// ---- VISUs/EtherCAT_Diag2.TcVIS
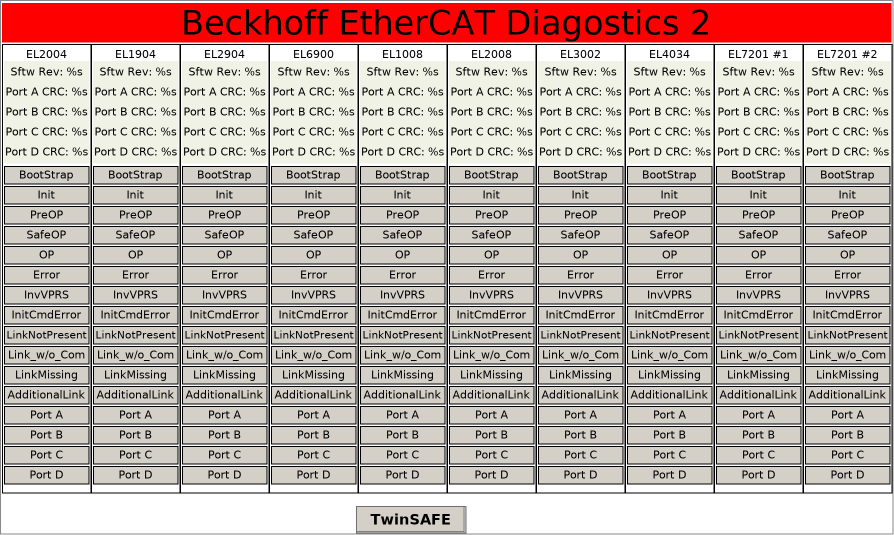
VISUALIZATION EtherCAT_Diag2  // 894x535
    Button (356,506 110x27), "TwinSAFE"
        OnMouseClick: change screen: TwinSAFE
    RoundedRectangle (2,3 889x39), "Beckhoff EtherCAT Diagostics 2"
    Group (2,42 89x451)
        RoundedRectangle (0,2 89x449)
        Label (2,0 85x25), "EL2004"
        Rectangle (2,19 85x22), "Sftw Rev: %s", text variable: g_iHMI_ProdCodeEL2004
        Rectangle (2,39 85x22), "Port A CRC: %s", text variable: g_stHMI_EL2004CrcErrorEx.portA
        Rectangle (2,59 85x22), "Port B CRC: %s", text variable: g_stHMI_EL2004CrcErrorEx.portB
        Rectangle (2,79 85x22), "Port C CRC: %s", text variable: g_stHMI_EL2004CrcErrorEx.portC
        Rectangle (2,99 85x22), "Port D CRC: %s", text variable: g_stHMI_EL2004CrcErrorEx.portD
        Rectangle (2,124 85x18), "BootStrap", colour toggle: g_stHMI_EL2004EcSlaveStateBits.bBootStrap
        Rectangle (2,144 85x18), "Init", colour toggle: g_stHMI_EL2004EcSlaveStateBits.bInit
        Rectangle (2,164 85x18), "PreOP", colour toggle: g_stHMI_EL2004EcSlaveStateBits.bPreop
        Rectangle (2,184 85x18), "SafeOP", colour toggle: g_stHMI_EL2004EcSlaveStateBits.bSafeOp
        Rectangle (2,204 85x18), "OP", colour toggle: g_stHMI_EL2004EcSlaveStateBits.bOp
        Rectangle (2,224 85x18), "Error", colour toggle: g_stHMI_EL2004EcSlaveStateBits.bError
        Rectangle (2,244 85x18), "InvVPRS", colour toggle: g_stHMI_EL2004EcSlaveStateBits.bInvVPRS
        Rectangle (2,264 85x18), "InitCmdError", colour toggle: g_stHMI_EL2004EcSlaveStateBits.bInitCmdError
        Rectangle (2,284 85x18), "LinkNotPresent", colour toggle: g_stHMI_EL2004EcSlaveStateBits.bLinkNotPresent
        Rectangle (2,304 85x18), "Link_w/o_Com", colour toggle: g_stHMI_EL2004EcSlaveStateBits.bLinkWithoutComm
        Rectangle (2,324 85x18), "LinkMissing", colour toggle: g_stHMI_EL2004EcSlaveStateBits.bLinkMissing
        Rectangle (2,344 85x18), "AdditionalLink", colour toggle: g_stHMI_EL2004EcSlaveStateBits.bAdditionalLink
        Rectangle (2,364 85x18), "Port A", colour toggle: g_stHMI_EL2004EcSlaveStateBits.bPortA
        Rectangle (2,384 85x18), "Port B", colour toggle: g_stHMI_EL2004EcSlaveStateBits.bPortB
        Rectangle (2,404 85x18), "Port C", colour toggle: g_stHMI_EL2004EcSlaveStateBits.bPortC
        Rectangle (2,424 85x18), "Port D", colour toggle: g_stHMI_EL2004EcSlaveStateBits.bPortD
    Group (91,42 89x451)
        RoundedRectangle (0,2 89x449)
        Label (2,0 85x25), "EL1904"
        Rectangle (2,19 85x22), "Sftw Rev: %s", text variable: g_iHMI_ProdCodeEL1904
        Rectangle (2,39 85x22), "Port A CRC: %s", text variable: g_stHMI_EL1904CrcErrorEx.portA
        Rectangle (2,59 85x22), "Port B CRC: %s", text variable: g_stHMI_EL1904CrcErrorEx.portB
        Rectangle (2,79 85x22), "Port C CRC: %s", text variable: g_stHMI_EL1904CrcErrorEx.portC
        Rectangle (2,99 85x22), "Port D CRC: %s", text variable: g_stHMI_EL1904CrcErrorEx.portD
        Rectangle (2,124 85x18), "BootStrap", colour toggle: g_stHMI_EL1904EcSlaveStateBits.bBootStrap
        Rectangle (2,144 85x18), "Init", colour toggle: g_stHMI_EL1904EcSlaveStateBits.bInit
        Rectangle (2,164 85x18), "PreOP", colour toggle: g_stHMI_EL1904EcSlaveStateBits.bPreop
        Rectangle (2,184 85x18), "SafeOP", colour toggle: g_stHMI_EL1904EcSlaveStateBits.bSafeOp
        Rectangle (2,204 85x18), "OP", colour toggle: g_stHMI_EL1904EcSlaveStateBits.bOp
        Rectangle (2,224 85x18), "Error", colour toggle: g_stHMI_EL1904EcSlaveStateBits.bError
        Rectangle (2,244 85x18), "InvVPRS", colour toggle: g_stHMI_EL1904EcSlaveStateBits.bInvVPRS
        Rectangle (2,264 85x18), "InitCmdError", colour toggle: g_stHMI_EL1904EcSlaveStateBits.bInitCmdError
        Rectangle (2,284 85x18), "LinkNotPresent", colour toggle: g_stHMI_EL1904EcSlaveStateBits.bLinkNotPresent
        Rectangle (2,304 85x18), "Link_w/o_Com", colour toggle: g_stHMI_EL1904EcSlaveStateBits.bLinkWithoutComm
        Rectangle (2,324 85x18), "LinkMissing", colour toggle: g_stHMI_EL1904EcSlaveStateBits.bLinkMissing
        Rectangle (2,344 85x18), "AdditionalLink", colour toggle: g_stHMI_EL1904EcSlaveStateBits.bAdditionalLink
        Rectangle (2,364 85x18), "Port A", colour toggle: g_stHMI_EL1904EcSlaveStateBits.bPortA
        Rectangle (2,384 85x18), "Port B", colour toggle: g_stHMI_EL1904EcSlaveStateBits.bPortB
        Rectangle (2,404 85x18), "Port C", colour toggle: g_stHMI_EL1904EcSlaveStateBits.bPortC
        Rectangle (2,424 85x18), "Port D", colour toggle: g_stHMI_EL1904EcSlaveStateBits.bPortD
    Group (180,42 89x451)
        RoundedRectangle (0,2 89x449)
        Label (2,0 85x25), "EL2904"
        Rectangle (2,19 85x22), "Sftw Rev: %s", text variable: g_iHMI_ProdCodeEL2904
        Rectangle (2,39 85x22), "Port A CRC: %s", text variable: g_stHMI_EL2904CrcErrorEx.portA
        Rectangle (2,59 85x22), "Port B CRC: %s", text variable: g_stHMI_EL2904CrcErrorEx.portB
        Rectangle (2,79 85x22), "Port C CRC: %s", text variable: g_stHMI_EL2904CrcErrorEx.portC
        Rectangle (2,99 85x22), "Port D CRC: %s", text variable: g_stHMI_EL2904CrcErrorEx.portD
        Rectangle (2,124 85x18), "BootStrap", colour toggle: g_stHMI_EL2904EcSlaveStateBits.bBootStrap
        Rectangle (2,144 85x18), "Init", colour toggle: g_stHMI_EL2904EcSlaveStateBits.bInit
        Rectangle (2,164 85x18), "PreOP", colour toggle: g_stHMI_EL2904EcSlaveStateBits.bPreop
        Rectangle (2,184 85x18), "SafeOP", colour toggle: g_stHMI_EL2904EcSlaveStateBits.bSafeOp
        Rectangle (2,204 85x18), "OP", colour toggle: g_stHMI_EL2904EcSlaveStateBits.bOp
        Rectangle (2,224 85x18), "Error", colour toggle: g_stHMI_EL2904EcSlaveStateBits.bError
        Rectangle (2,244 85x18), "InvVPRS", colour toggle: g_stHMI_EL2904EcSlaveStateBits.bInvVPRS
        Rectangle (2,264 85x18), "InitCmdError", colour toggle: g_stHMI_EL2904EcSlaveStateBits.bInitCmdError
        Rectangle (2,284 85x18), "LinkNotPresent", colour toggle: g_stHMI_EL2904EcSlaveStateBits.bLinkNotPresent
        Rectangle (2,304 85x18), "Link_w/o_Com", colour toggle: g_stHMI_EL2904EcSlaveStateBits.bLinkWithoutComm
        Rectangle (2,324 85x18), "LinkMissing", colour toggle: g_stHMI_EL2904EcSlaveStateBits.bLinkMissing
        Rectangle (2,344 85x18), "AdditionalLink", colour toggle: g_stHMI_EL2904EcSlaveStateBits.bAdditionalLink
        Rectangle (2,364 85x18), "Port A", colour toggle: g_stHMI_EL2904EcSlaveStateBits.bPortA
        Rectangle (2,384 85x18), "Port B", colour toggle: g_stHMI_EL2904EcSlaveStateBits.bPortB
        Rectangle (2,404 85x18), "Port C", colour toggle: g_stHMI_EL2904EcSlaveStateBits.bPortC
        Rectangle (2,424 85x18), "Port D", colour toggle: g_stHMI_EL2904EcSlaveStateBits.bPortD
    Group (269,42 89x451)
        RoundedRectangle (0,2 89x449)
        Label (2,0 85x25), "EL6900"
        Rectangle (2,19 85x22), "Sftw Rev: %s", text variable: g_iHMI_ProdCodeEL6900
        Rectangle (2,39 85x22), "Port A CRC: %s", text variable: g_stHMI_EL6900CrcErrorEx.portA
        Rectangle (2,59 85x22), "Port B CRC: %s", text variable: g_stHMI_EL6900CrcErrorEx.portB
        Rectangle (2,79 85x22), "Port C CRC: %s", text variable: g_stHMI_EL6900CrcErrorEx.portC
        Rectangle (2,99 85x22), "Port D CRC: %s", text variable: g_stHMI_EL6900CrcErrorEx.portD
        Rectangle (2,124 85x18), "BootStrap", colour toggle: g_stHMI_EL6900EcSlaveStateBits.bBootStrap
        Rectangle (2,144 85x18), "Init", colour toggle: g_stHMI_EL6900EcSlaveStateBits.bInit
        Rectangle (2,164 85x18), "PreOP", colour toggle: g_stHMI_EL6900EcSlaveStateBits.bPreop
        Rectangle (2,184 85x18), "SafeOP", colour toggle: g_stHMI_EL6900EcSlaveStateBits.bSafeOp
        Rectangle (2,204 85x18), "OP", colour toggle: g_stHMI_EL6900EcSlaveStateBits.bOp
        Rectangle (2,224 85x18), "Error", colour toggle: g_stHMI_EL6900EcSlaveStateBits.bError
        Rectangle (2,244 85x18), "InvVPRS", colour toggle: g_stHMI_EL6900EcSlaveStateBits.bInvVPRS
        Rectangle (2,264 85x18), "InitCmdError", colour toggle: g_stHMI_EL6900EcSlaveStateBits.bInitCmdError
        Rectangle (2,284 85x18), "LinkNotPresent", colour toggle: g_stHMI_EL6900EcSlaveStateBits.bLinkNotPresent
        Rectangle (2,304 85x18), "Link_w/o_Com", colour toggle: g_stHMI_EL6900EcSlaveStateBits.bLinkWithoutComm
        Rectangle (2,324 85x18), "LinkMissing", colour toggle: g_stHMI_EL6900EcSlaveStateBits.bLinkMissing
        Rectangle (2,344 85x18), "AdditionalLink", colour toggle: g_stHMI_EL6900EcSlaveStateBits.bAdditionalLink
        Rectangle (2,364 85x18), "Port A", colour toggle: g_stHMI_EL6900EcSlaveStateBits.bPortA
        Rectangle (2,384 85x18), "Port B", colour toggle: g_stHMI_EL6900EcSlaveStateBits.bPortB
        Rectangle (2,404 85x18), "Port C", colour toggle: g_stHMI_EL6900EcSlaveStateBits.bPortC
        Rectangle (2,424 85x18), "Port D", colour toggle: g_stHMI_EL6900EcSlaveStateBits.bPortD
    Group (358,42 89x451)
        RoundedRectangle (0,2 89x449)
        Label (2,0 85x25), "EL1008"
        Rectangle (2,19 85x22), "Sftw Rev: %s", text variable: g_iHMI_ProdCodeEL1008
        Rectangle (2,39 85x22), "Port A CRC: %s", text variable: g_stHMI_EL1008CrcErrorEx.portA
        Rectangle (2,59 85x22), "Port B CRC: %s", text variable: g_stHMI_EL1008CrcErrorEx.portB
        Rectangle (2,79 85x22), "Port C CRC: %s", text variable: g_stHMI_EL1008CrcErrorEx.portC
        Rectangle (2,99 85x22), "Port D CRC: %s", text variable: g_stHMI_EL1008CrcErrorEx.portD
        Rectangle (2,124 85x18), "BootStrap", colour toggle: g_stHMI_EL1008EcSlaveStateBits.bBootStrap
        Rectangle (2,144 85x18), "Init", colour toggle: g_stHMI_EL1008EcSlaveStateBits.bInit
        Rectangle (2,164 85x18), "PreOP", colour toggle: g_stHMI_EL1008EcSlaveStateBits.bPreop
        Rectangle (2,184 85x18), "SafeOP", colour toggle: g_stHMI_EL1008EcSlaveStateBits.bSafeOp
        Rectangle (2,204 85x18), "OP", colour toggle: g_stHMI_EL1008EcSlaveStateBits.bOp
        Rectangle (2,224 85x18), "Error", colour toggle: g_stHMI_EL1008EcSlaveStateBits.bError
        Rectangle (2,244 85x18), "InvVPRS", colour toggle: g_stHMI_EL1008EcSlaveStateBits.bInvVPRS
        Rectangle (2,264 85x18), "InitCmdError", colour toggle: g_stHMI_EL1008EcSlaveStateBits.bInitCmdError
        Rectangle (2,284 85x18), "LinkNotPresent", colour toggle: g_stHMI_EL1008EcSlaveStateBits.bLinkNotPresent
        Rectangle (2,304 85x18), "Link_w/o_Com", colour toggle: g_stHMI_EL1008EcSlaveStateBits.bLinkWithoutComm
        Rectangle (2,324 85x18), "LinkMissing", colour toggle: g_stHMI_EL1008EcSlaveStateBits.bLinkMissing
        Rectangle (2,344 85x18), "AdditionalLink", colour toggle: g_stHMI_EL1008EcSlaveStateBits.bAdditionalLink
        Rectangle (2,364 85x18), "Port A", colour toggle: g_stHMI_EL1008EcSlaveStateBits.bPortA
        Rectangle (2,384 85x18), "Port B", colour toggle: g_stHMI_EL1008EcSlaveStateBits.bPortB
        Rectangle (2,404 85x18), "Port C", colour toggle: g_stHMI_EL1008EcSlaveStateBits.bPortC
        Rectangle (2,424 85x18), "Port D", colour toggle: g_stHMI_EL1008EcSlaveStateBits.bPortD
    Group (447,42 89x451)
        RoundedRectangle (0,2 89x449)
        Label (2,0 85x25), "EL2008"
        Rectangle (2,19 85x22), "Sftw Rev: %s", text variable: g_iHMI_ProdCodeEL2008
        Rectangle (2,39 85x22), "Port A CRC: %s", text variable: g_stHMI_EL2008CrcErrorEx.portA
        Rectangle (2,59 85x22), "Port B CRC: %s", text variable: g_stHMI_EL2008CrcErrorEx.portB
        Rectangle (2,79 85x22), "Port C CRC: %s", text variable: g_stHMI_EL2008CrcErrorEx.portC
        Rectangle (2,99 85x22), "Port D CRC: %s", text variable: g_stHMI_EL2008CrcErrorEx.portD
        Rectangle (2,124 85x18), "BootStrap", colour toggle: g_stHMI_EL2008EcSlaveStateBits.bBootStrap
        Rectangle (2,144 85x18), "Init", colour toggle: g_stHMI_EL2008EcSlaveStateBits.bInit
        Rectangle (2,164 85x18), "PreOP", colour toggle: g_stHMI_EL2008EcSlaveStateBits.bPreop
        Rectangle (2,184 85x18), "SafeOP", colour toggle: g_stHMI_EL2008EcSlaveStateBits.bSafeOp
        Rectangle (2,204 85x18), "OP", colour toggle: g_stHMI_EL2008EcSlaveStateBits.bOp
        Rectangle (2,224 85x18), "Error", colour toggle: g_stHMI_EL2008EcSlaveStateBits.bError
        Rectangle (2,244 85x18), "InvVPRS", colour toggle: g_stHMI_EL2008EcSlaveStateBits.bInvVPRS
        Rectangle (2,264 85x18), "InitCmdError", colour toggle: g_stHMI_EL2008EcSlaveStateBits.bInitCmdError
        Rectangle (2,284 85x18), "LinkNotPresent", colour toggle: g_stHMI_EL2008EcSlaveStateBits.bLinkNotPresent
        Rectangle (2,304 85x18), "Link_w/o_Com", colour toggle: g_stHMI_EL2008EcSlaveStateBits.bLinkWithoutComm
        Rectangle (2,324 85x18), "LinkMissing", colour toggle: g_stHMI_EL2008EcSlaveStateBits.bLinkMissing
        Rectangle (2,344 85x18), "AdditionalLink", colour toggle: g_stHMI_EL2008EcSlaveStateBits.bAdditionalLink
        Rectangle (2,364 85x18), "Port A", colour toggle: g_stHMI_EL2008EcSlaveStateBits.bPortA
        Rectangle (2,384 85x18), "Port B", colour toggle: g_stHMI_EL2008EcSlaveStateBits.bPortB
        Rectangle (2,404 85x18), "Port C", colour toggle: g_stHMI_EL2008EcSlaveStateBits.bPortC
        Rectangle (2,424 85x18), "Port D", colour toggle: g_stHMI_EL2008EcSlaveStateBits.bPortD
    Group (536,42 89x451)
        RoundedRectangle (0,2 89x449)
        Label (2,0 85x25), "EL3002"
        Rectangle (2,19 85x22), "Sftw Rev: %s", text variable: g_iHMI_ProdCodeEL3002
        Rectangle (2,39 85x22), "Port A CRC: %s", text variable: g_stHMI_EL3002CrcErrorEx.portA
        Rectangle (2,59 85x22), "Port B CRC: %s", text variable: g_stHMI_EL3002CrcErrorEx.portB
        Rectangle (2,79 85x22), "Port C CRC: %s", text variable: g_stHMI_EL3002CrcErrorEx.portC
        Rectangle (2,99 85x22), "Port D CRC: %s", text variable: g_stHMI_EL3002CrcErrorEx.portD
        Rectangle (2,124 85x18), "BootStrap", colour toggle: g_stHMI_EL3002EcSlaveStateBits.bBootStrap
        Rectangle (2,144 85x18), "Init", colour toggle: g_stHMI_EL3002EcSlaveStateBits.bInit
        Rectangle (2,164 85x18), "PreOP", colour toggle: g_stHMI_EL3002EcSlaveStateBits.bPreop
        Rectangle (2,184 85x18), "SafeOP", colour toggle: g_stHMI_EL3002EcSlaveStateBits.bSafeOp
        Rectangle (2,204 85x18), "OP", colour toggle: g_stHMI_EL3002EcSlaveStateBits.bOp
        Rectangle (2,224 85x18), "Error", colour toggle: g_stHMI_EL3002EcSlaveStateBits.bError
        Rectangle (2,244 85x18), "InvVPRS", colour toggle: g_stHMI_EL3002EcSlaveStateBits.bInvVPRS
        Rectangle (2,264 85x18), "InitCmdError", colour toggle: g_stHMI_EL3002EcSlaveStateBits.bInitCmdError
        Rectangle (2,284 85x18), "LinkNotPresent", colour toggle: g_stHMI_EL3002EcSlaveStateBits.bLinkNotPresent
        Rectangle (2,304 85x18), "Link_w/o_Com", colour toggle: g_stHMI_EL3002EcSlaveStateBits.bLinkWithoutComm
        Rectangle (2,324 85x18), "LinkMissing", colour toggle: g_stHMI_EL3002EcSlaveStateBits.bLinkMissing
        Rectangle (2,344 85x18), "AdditionalLink", colour toggle: g_stHMI_EL3002EcSlaveStateBits.bAdditionalLink
        Rectangle (2,364 85x18), "Port A", colour toggle: g_stHMI_EL3002EcSlaveStateBits.bPortA
        Rectangle (2,384 85x18), "Port B", colour toggle: g_stHMI_EL3002EcSlaveStateBits.bPortB
        Rectangle (2,404 85x18), "Port C", colour toggle: g_stHMI_EL3002EcSlaveStateBits.bPortC
        Rectangle (2,424 85x18), "Port D", colour toggle: g_stHMI_EL3002EcSlaveStateBits.bPortD
    Group (625,42 89x451)
        RoundedRectangle (0,2 89x449)
        Label (2,0 85x25), "EL4034"
        Rectangle (2,19 85x22), "Sftw Rev: %s", text variable: g_iHMI_ProdCodeEL4034
        Rectangle (2,39 85x22), "Port A CRC: %s", text variable: g_stHMI_EL4034CrcErrorEx.portA
        Rectangle (2,59 85x22), "Port B CRC: %s", text variable: g_stHMI_EL4034CrcErrorEx.portB
        Rectangle (2,79 85x22), "Port C CRC: %s", text variable: g_stHMI_EL4034CrcErrorEx.portC
        Rectangle (2,99 85x22), "Port D CRC: %s", text variable: g_stHMI_EL4034CrcErrorEx.portD
        Rectangle (2,124 85x18), "BootStrap", colour toggle: g_stHMI_EL4034EcSlaveStateBits.bBootStrap
        Rectangle (2,144 85x18), "Init", colour toggle: g_stHMI_EL4034EcSlaveStateBits.bInit
        Rectangle (2,164 85x18), "PreOP", colour toggle: g_stHMI_EL4034EcSlaveStateBits.bPreop
        Rectangle (2,184 85x18), "SafeOP", colour toggle: g_stHMI_EL4034EcSlaveStateBits.bSafeOp
        Rectangle (2,204 85x18), "OP", colour toggle: g_stHMI_EL4034EcSlaveStateBits.bOp
        Rectangle (2,224 85x18), "Error", colour toggle: g_stHMI_EL4034EcSlaveStateBits.bError
        Rectangle (2,244 85x18), "InvVPRS", colour toggle: g_stHMI_EL4034EcSlaveStateBits.bInvVPRS
        Rectangle (2,264 85x18), "InitCmdError", colour toggle: g_stHMI_EL4034EcSlaveStateBits.bInitCmdError
        Rectangle (2,284 85x18), "LinkNotPresent", colour toggle: g_stHMI_EL4034EcSlaveStateBits.bLinkNotPresent
        Rectangle (2,304 85x18), "Link_w/o_Com", colour toggle: g_stHMI_EL4034EcSlaveStateBits.bLinkWithoutComm
        Rectangle (2,324 85x18), "LinkMissing", colour toggle: g_stHMI_EL4034EcSlaveStateBits.bLinkMissing
        Rectangle (2,344 85x18), "AdditionalLink", colour toggle: g_stHMI_EL4034EcSlaveStateBits.bAdditionalLink
        Rectangle (2,364 85x18), "Port A", colour toggle: g_stHMI_EL4034EcSlaveStateBits.bPortA
        Rectangle (2,384 85x18), "Port B", colour toggle: g_stHMI_EL4034EcSlaveStateBits.bPortB
        Rectangle (2,404 85x18), "Port C", colour toggle: g_stHMI_EL4034EcSlaveStateBits.bPortC
        Rectangle (2,424 85x18), "Port D", colour toggle: g_stHMI_EL4034EcSlaveStateBits.bPortD
    Group (714,42 89x451)
        RoundedRectangle (0,2 89x449)
        Label (2,0 85x25), "EL7201 #1"
        Rectangle (2,19 85x22), "Sftw Rev: %s", text variable: g_iHMI_ProdCodeEL7201_1
        Rectangle (2,39 85x22), "Port A CRC: %s", text variable: g_stHMI_EL7201_1CrcErrorEx.portA
        Rectangle (2,59 85x22), "Port B CRC: %s", text variable: g_stHMI_EL7201_1CrcErrorEx.portB
        Rectangle (2,79 85x22), "Port C CRC: %s", text variable: g_stHMI_EL7201_1CrcErrorEx.portC
        Rectangle (2,99 85x22), "Port D CRC: %s", text variable: g_stHMI_EL7201_1CrcErrorEx.portD
        Rectangle (2,124 85x18), "BootStrap", colour toggle: g_stHMI_EL7201_1EcSlaveStateBits.bBootStrap
        Rectangle (2,144 85x18), "Init", colour toggle: g_stHMI_EL7201_1EcSlaveStateBits.bInit
        Rectangle (2,164 85x18), "PreOP", colour toggle: g_stHMI_EL7201_1EcSlaveStateBits.bPreop
        Rectangle (2,184 85x18), "SafeOP", colour toggle: g_stHMI_EL7201_1EcSlaveStateBits.bSafeOp
        Rectangle (2,204 85x18), "OP", colour toggle: g_stHMI_EL7201_1EcSlaveStateBits.bOp
        Rectangle (2,224 85x18), "Error", colour toggle: g_stHMI_EL7201_1EcSlaveStateBits.bError
        Rectangle (2,244 85x18), "InvVPRS", colour toggle: g_stHMI_EL7201_1EcSlaveStateBits.bInvVPRS
        Rectangle (2,264 85x18), "InitCmdError", colour toggle: g_stHMI_EL7201_1EcSlaveStateBits.bInitCmdError
        Rectangle (2,284 85x18), "LinkNotPresent", colour toggle: g_stHMI_EL7201_1EcSlaveStateBits.bLinkNotPresent
        Rectangle (2,304 85x18), "Link_w/o_Com", colour toggle: g_stHMI_EL7201_1EcSlaveStateBits.bLinkWithoutComm
        Rectangle (2,324 85x18), "LinkMissing", colour toggle: g_stHMI_EL7201_1EcSlaveStateBits.bLinkMissing
        Rectangle (2,344 85x18), "AdditionalLink", colour toggle: g_stHMI_EL7201_1EcSlaveStateBits.bAdditionalLink
        Rectangle (2,364 85x18), "Port A", colour toggle: g_stHMI_EL7201_1EcSlaveStateBits.bPortA
        Rectangle (2,384 85x18), "Port B", colour toggle: g_stHMI_EL7201_1EcSlaveStateBits.bPortB
        Rectangle (2,404 85x18), "Port C", colour toggle: g_stHMI_EL7201_1EcSlaveStateBits.bPortC
        Rectangle (2,424 85x18), "Port D", colour toggle: g_stHMI_EL7201_1EcSlaveStateBits.bPortD
    Group (803,42 89x451)
        RoundedRectangle (0,2 89x449)
        Label (2,0 85x25), "EL7201 #2"
        Rectangle (2,19 85x22), "Sftw Rev: %s", text variable: g_iHMI_ProdCodeEL7201_2
        Rectangle (2,39 85x22), "Port A CRC: %s", text variable: g_stHMI_EL7201_2CrcErrorEx.portA
        Rectangle (2,59 85x22), "Port B CRC: %s", text variable: g_stHMI_EL7201_2CrcErrorEx.portB
        Rectangle (2,79 85x22), "Port C CRC: %s", text variable: g_stHMI_EL7201_2CrcErrorEx.portC
        Rectangle (2,99 85x22), "Port D CRC: %s", text variable: g_stHMI_EL7201_2CrcErrorEx.portD
        Rectangle (2,124 85x18), "BootStrap", colour toggle: g_stHMI_EL7201_2EcSlaveStateBits.bBootStrap
        Rectangle (2,144 85x18), "Init", colour toggle: g_stHMI_EL7201_2EcSlaveStateBits.bInit
        Rectangle (2,164 85x18), "PreOP", colour toggle: g_stHMI_EL7201_2EcSlaveStateBits.bPreop
        Rectangle (2,184 85x18), "SafeOP", colour toggle: g_stHMI_EL7201_2EcSlaveStateBits.bSafeOp
        Rectangle (2,204 85x18), "OP", colour toggle: g_stHMI_EL7201_2EcSlaveStateBits.bOp
        Rectangle (2,224 85x18), "Error", colour toggle: g_stHMI_EL7201_2EcSlaveStateBits.bError
        Rectangle (2,244 85x18), "InvVPRS", colour toggle: g_stHMI_EL7201_2EcSlaveStateBits.bInvVPRS
        Rectangle (2,264 85x18), "InitCmdError", colour toggle: g_stHMI_EL7201_2EcSlaveStateBits.bInitCmdError
        Rectangle (2,284 85x18), "LinkNotPresent", colour toggle: g_stHMI_EL7201_2EcSlaveStateBits.bLinkNotPresent
        Rectangle (2,304 85x18), "Link_w/o_Com", colour toggle: g_stHMI_EL7201_2EcSlaveStateBits.bLinkWithoutComm
        Rectangle (2,324 85x18), "LinkMissing", colour toggle: g_stHMI_EL7201_2EcSlaveStateBits.bLinkMissing
        Rectangle (2,344 85x18), "AdditionalLink", colour toggle: g_stHMI_EL7201_2EcSlaveStateBits.bAdditionalLink
        Rectangle (2,364 85x18), "Port A", colour toggle: g_stHMI_EL7201_2EcSlaveStateBits.bPortA
        Rectangle (2,384 85x18), "Port B", colour toggle: g_stHMI_EL7201_2EcSlaveStateBits.bPortB
        Rectangle (2,404 85x18), "Port C", colour toggle: g_stHMI_EL7201_2EcSlaveStateBits.bPortC
        Rectangle (2,424 85x18), "Port D", colour toggle: g_stHMI_EL7201_2EcSlaveStateBits.bPortD
END_VISUALIZATION

// ---- VISUs/EtherCAT_Diag2.TcVIS
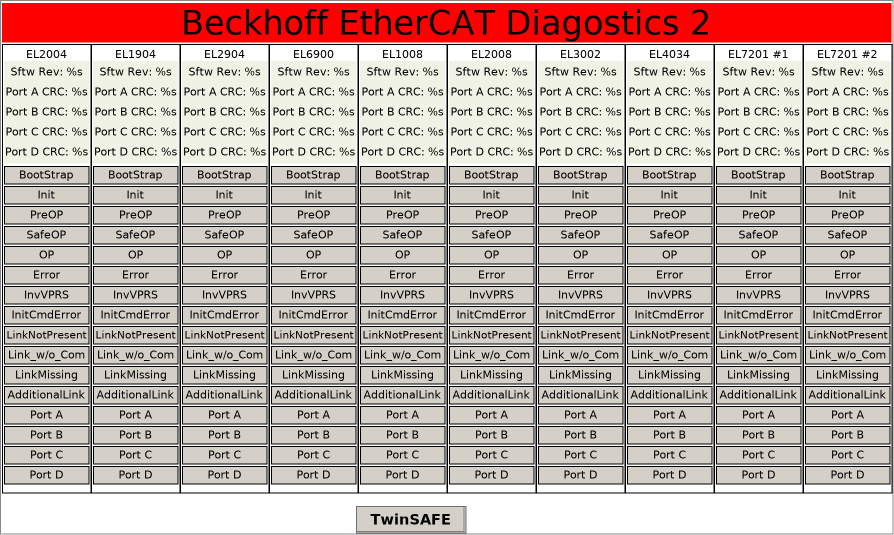
VISUALIZATION EtherCAT_Diag2  // 894x535
    Button (356,506 110x27), "TwinSAFE"
        OnMouseClick: change screen: TwinSAFE
    RoundedRectangle (2,3 889x39), "Beckhoff EtherCAT Diagostics 2"
    Group (2,42 89x451)
        RoundedRectangle (0,2 89x449)
        Label (2,0 85x25), "EL2004"
        Rectangle (2,19 85x22), "Sftw Rev: %s", text variable: g_iHMI_ProdCodeEL2004
        Rectangle (2,39 85x22), "Port A CRC: %s", text variable: g_stHMI_EL2004CrcErrorEx.portA
        Rectangle (2,59 85x22), "Port B CRC: %s", text variable: g_stHMI_EL2004CrcErrorEx.portB
        Rectangle (2,79 85x22), "Port C CRC: %s", text variable: g_stHMI_EL2004CrcErrorEx.portC
        Rectangle (2,99 85x22), "Port D CRC: %s", text variable: g_stHMI_EL2004CrcErrorEx.portD
        Rectangle (2,124 85x18), "BootStrap", colour toggle: g_stHMI_EL2004EcSlaveStateBits.bBootStrap
        Rectangle (2,144 85x18), "Init", colour toggle: g_stHMI_EL2004EcSlaveStateBits.bInit
        Rectangle (2,164 85x18), "PreOP", colour toggle: g_stHMI_EL2004EcSlaveStateBits.bPreop
        Rectangle (2,184 85x18), "SafeOP", colour toggle: g_stHMI_EL2004EcSlaveStateBits.bSafeOp
        Rectangle (2,204 85x18), "OP", colour toggle: g_stHMI_EL2004EcSlaveStateBits.bOp
        Rectangle (2,224 85x18), "Error", colour toggle: g_stHMI_EL2004EcSlaveStateBits.bError
        Rectangle (2,244 85x18), "InvVPRS", colour toggle: g_stHMI_EL2004EcSlaveStateBits.bInvVPRS
        Rectangle (2,264 85x18), "InitCmdError", colour toggle: g_stHMI_EL2004EcSlaveStateBits.bInitCmdError
        Rectangle (2,284 85x18), "LinkNotPresent", colour toggle: g_stHMI_EL2004EcSlaveStateBits.bLinkNotPresent
        Rectangle (2,304 85x18), "Link_w/o_Com", colour toggle: g_stHMI_EL2004EcSlaveStateBits.bLinkWithoutComm
        Rectangle (2,324 85x18), "LinkMissing", colour toggle: g_stHMI_EL2004EcSlaveStateBits.bLinkMissing
        Rectangle (2,344 85x18), "AdditionalLink", colour toggle: g_stHMI_EL2004EcSlaveStateBits.bAdditionalLink
        Rectangle (2,364 85x18), "Port A", colour toggle: g_stHMI_EL2004EcSlaveStateBits.bPortA
        Rectangle (2,384 85x18), "Port B", colour toggle: g_stHMI_EL2004EcSlaveStateBits.bPortB
        Rectangle (2,404 85x18), "Port C", colour toggle: g_stHMI_EL2004EcSlaveStateBits.bPortC
        Rectangle (2,424 85x18), "Port D", colour toggle: g_stHMI_EL2004EcSlaveStateBits.bPortD
    Group (91,42 89x451)
        RoundedRectangle (0,2 89x449)
        Label (2,0 85x25), "EL1904"
        Rectangle (2,19 85x22), "Sftw Rev: %s", text variable: g_iHMI_ProdCodeEL1904
        Rectangle (2,39 85x22), "Port A CRC: %s", text variable: g_stHMI_EL1904CrcErrorEx.portA
        Rectangle (2,59 85x22), "Port B CRC: %s", text variable: g_stHMI_EL1904CrcErrorEx.portB
        Rectangle (2,79 85x22), "Port C CRC: %s", text variable: g_stHMI_EL1904CrcErrorEx.portC
        Rectangle (2,99 85x22), "Port D CRC: %s", text variable: g_stHMI_EL1904CrcErrorEx.portD
        Rectangle (2,124 85x18), "BootStrap", colour toggle: g_stHMI_EL1904EcSlaveStateBits.bBootStrap
        Rectangle (2,144 85x18), "Init", colour toggle: g_stHMI_EL1904EcSlaveStateBits.bInit
        Rectangle (2,164 85x18), "PreOP", colour toggle: g_stHMI_EL1904EcSlaveStateBits.bPreop
        Rectangle (2,184 85x18), "SafeOP", colour toggle: g_stHMI_EL1904EcSlaveStateBits.bSafeOp
        Rectangle (2,204 85x18), "OP", colour toggle: g_stHMI_EL1904EcSlaveStateBits.bOp
        Rectangle (2,224 85x18), "Error", colour toggle: g_stHMI_EL1904EcSlaveStateBits.bError
        Rectangle (2,244 85x18), "InvVPRS", colour toggle: g_stHMI_EL1904EcSlaveStateBits.bInvVPRS
        Rectangle (2,264 85x18), "InitCmdError", colour toggle: g_stHMI_EL1904EcSlaveStateBits.bInitCmdError
        Rectangle (2,284 85x18), "LinkNotPresent", colour toggle: g_stHMI_EL1904EcSlaveStateBits.bLinkNotPresent
        Rectangle (2,304 85x18), "Link_w/o_Com", colour toggle: g_stHMI_EL1904EcSlaveStateBits.bLinkWithoutComm
        Rectangle (2,324 85x18), "LinkMissing", colour toggle: g_stHMI_EL1904EcSlaveStateBits.bLinkMissing
        Rectangle (2,344 85x18), "AdditionalLink", colour toggle: g_stHMI_EL1904EcSlaveStateBits.bAdditionalLink
        Rectangle (2,364 85x18), "Port A", colour toggle: g_stHMI_EL1904EcSlaveStateBits.bPortA
        Rectangle (2,384 85x18), "Port B", colour toggle: g_stHMI_EL1904EcSlaveStateBits.bPortB
        Rectangle (2,404 85x18), "Port C", colour toggle: g_stHMI_EL1904EcSlaveStateBits.bPortC
        Rectangle (2,424 85x18), "Port D", colour toggle: g_stHMI_EL1904EcSlaveStateBits.bPortD
    Group (180,42 89x451)
        RoundedRectangle (0,2 89x449)
        Label (2,0 85x25), "EL2904"
        Rectangle (2,19 85x22), "Sftw Rev: %s", text variable: g_iHMI_ProdCodeEL2904
        Rectangle (2,39 85x22), "Port A CRC: %s", text variable: g_stHMI_EL2904CrcErrorEx.portA
        Rectangle (2,59 85x22), "Port B CRC: %s", text variable: g_stHMI_EL2904CrcErrorEx.portB
        Rectangle (2,79 85x22), "Port C CRC: %s", text variable: g_stHMI_EL2904CrcErrorEx.portC
        Rectangle (2,99 85x22), "Port D CRC: %s", text variable: g_stHMI_EL2904CrcErrorEx.portD
        Rectangle (2,124 85x18), "BootStrap", colour toggle: g_stHMI_EL2904EcSlaveStateBits.bBootStrap
        Rectangle (2,144 85x18), "Init", colour toggle: g_stHMI_EL2904EcSlaveStateBits.bInit
        Rectangle (2,164 85x18), "PreOP", colour toggle: g_stHMI_EL2904EcSlaveStateBits.bPreop
        Rectangle (2,184 85x18), "SafeOP", colour toggle: g_stHMI_EL2904EcSlaveStateBits.bSafeOp
        Rectangle (2,204 85x18), "OP", colour toggle: g_stHMI_EL2904EcSlaveStateBits.bOp
        Rectangle (2,224 85x18), "Error", colour toggle: g_stHMI_EL2904EcSlaveStateBits.bError
        Rectangle (2,244 85x18), "InvVPRS", colour toggle: g_stHMI_EL2904EcSlaveStateBits.bInvVPRS
        Rectangle (2,264 85x18), "InitCmdError", colour toggle: g_stHMI_EL2904EcSlaveStateBits.bInitCmdError
        Rectangle (2,284 85x18), "LinkNotPresent", colour toggle: g_stHMI_EL2904EcSlaveStateBits.bLinkNotPresent
        Rectangle (2,304 85x18), "Link_w/o_Com", colour toggle: g_stHMI_EL2904EcSlaveStateBits.bLinkWithoutComm
        Rectangle (2,324 85x18), "LinkMissing", colour toggle: g_stHMI_EL2904EcSlaveStateBits.bLinkMissing
        Rectangle (2,344 85x18), "AdditionalLink", colour toggle: g_stHMI_EL2904EcSlaveStateBits.bAdditionalLink
        Rectangle (2,364 85x18), "Port A", colour toggle: g_stHMI_EL2904EcSlaveStateBits.bPortA
        Rectangle (2,384 85x18), "Port B", colour toggle: g_stHMI_EL2904EcSlaveStateBits.bPortB
        Rectangle (2,404 85x18), "Port C", colour toggle: g_stHMI_EL2904EcSlaveStateBits.bPortC
        Rectangle (2,424 85x18), "Port D", colour toggle: g_stHMI_EL2904EcSlaveStateBits.bPortD
    Group (269,42 89x451)
        RoundedRectangle (0,2 89x449)
        Label (2,0 85x25), "EL6900"
        Rectangle (2,19 85x22), "Sftw Rev: %s", text variable: g_iHMI_ProdCodeEL6900
        Rectangle (2,39 85x22), "Port A CRC: %s", text variable: g_stHMI_EL6900CrcErrorEx.portA
        Rectangle (2,59 85x22), "Port B CRC: %s", text variable: g_stHMI_EL6900CrcErrorEx.portB
        Rectangle (2,79 85x22), "Port C CRC: %s", text variable: g_stHMI_EL6900CrcErrorEx.portC
        Rectangle (2,99 85x22), "Port D CRC: %s", text variable: g_stHMI_EL6900CrcErrorEx.portD
        Rectangle (2,124 85x18), "BootStrap", colour toggle: g_stHMI_EL6900EcSlaveStateBits.bBootStrap
        Rectangle (2,144 85x18), "Init", colour toggle: g_stHMI_EL6900EcSlaveStateBits.bInit
        Rectangle (2,164 85x18), "PreOP", colour toggle: g_stHMI_EL6900EcSlaveStateBits.bPreop
        Rectangle (2,184 85x18), "SafeOP", colour toggle: g_stHMI_EL6900EcSlaveStateBits.bSafeOp
        Rectangle (2,204 85x18), "OP", colour toggle: g_stHMI_EL6900EcSlaveStateBits.bOp
        Rectangle (2,224 85x18), "Error", colour toggle: g_stHMI_EL6900EcSlaveStateBits.bError
        Rectangle (2,244 85x18), "InvVPRS", colour toggle: g_stHMI_EL6900EcSlaveStateBits.bInvVPRS
        Rectangle (2,264 85x18), "InitCmdError", colour toggle: g_stHMI_EL6900EcSlaveStateBits.bInitCmdError
        Rectangle (2,284 85x18), "LinkNotPresent", colour toggle: g_stHMI_EL6900EcSlaveStateBits.bLinkNotPresent
        Rectangle (2,304 85x18), "Link_w/o_Com", colour toggle: g_stHMI_EL6900EcSlaveStateBits.bLinkWithoutComm
        Rectangle (2,324 85x18), "LinkMissing", colour toggle: g_stHMI_EL6900EcSlaveStateBits.bLinkMissing
        Rectangle (2,344 85x18), "AdditionalLink", colour toggle: g_stHMI_EL6900EcSlaveStateBits.bAdditionalLink
        Rectangle (2,364 85x18), "Port A", colour toggle: g_stHMI_EL6900EcSlaveStateBits.bPortA
        Rectangle (2,384 85x18), "Port B", colour toggle: g_stHMI_EL6900EcSlaveStateBits.bPortB
        Rectangle (2,404 85x18), "Port C", colour toggle: g_stHMI_EL6900EcSlaveStateBits.bPortC
        Rectangle (2,424 85x18), "Port D", colour toggle: g_stHMI_EL6900EcSlaveStateBits.bPortD
    Group (358,42 89x451)
        RoundedRectangle (0,2 89x449)
        Label (2,0 85x25), "EL1008"
        Rectangle (2,19 85x22), "Sftw Rev: %s", text variable: g_iHMI_ProdCodeEL1008
        Rectangle (2,39 85x22), "Port A CRC: %s", text variable: g_stHMI_EL1008CrcErrorEx.portA
        Rectangle (2,59 85x22), "Port B CRC: %s", text variable: g_stHMI_EL1008CrcErrorEx.portB
        Rectangle (2,79 85x22), "Port C CRC: %s", text variable: g_stHMI_EL1008CrcErrorEx.portC
        Rectangle (2,99 85x22), "Port D CRC: %s", text variable: g_stHMI_EL1008CrcErrorEx.portD
        Rectangle (2,124 85x18), "BootStrap", colour toggle: g_stHMI_EL1008EcSlaveStateBits.bBootStrap
        Rectangle (2,144 85x18), "Init", colour toggle: g_stHMI_EL1008EcSlaveStateBits.bInit
        Rectangle (2,164 85x18), "PreOP", colour toggle: g_stHMI_EL1008EcSlaveStateBits.bPreop
        Rectangle (2,184 85x18), "SafeOP", colour toggle: g_stHMI_EL1008EcSlaveStateBits.bSafeOp
        Rectangle (2,204 85x18), "OP", colour toggle: g_stHMI_EL1008EcSlaveStateBits.bOp
        Rectangle (2,224 85x18), "Error", colour toggle: g_stHMI_EL1008EcSlaveStateBits.bError
        Rectangle (2,244 85x18), "InvVPRS", colour toggle: g_stHMI_EL1008EcSlaveStateBits.bInvVPRS
        Rectangle (2,264 85x18), "InitCmdError", colour toggle: g_stHMI_EL1008EcSlaveStateBits.bInitCmdError
        Rectangle (2,284 85x18), "LinkNotPresent", colour toggle: g_stHMI_EL1008EcSlaveStateBits.bLinkNotPresent
        Rectangle (2,304 85x18), "Link_w/o_Com", colour toggle: g_stHMI_EL1008EcSlaveStateBits.bLinkWithoutComm
        Rectangle (2,324 85x18), "LinkMissing", colour toggle: g_stHMI_EL1008EcSlaveStateBits.bLinkMissing
        Rectangle (2,344 85x18), "AdditionalLink", colour toggle: g_stHMI_EL1008EcSlaveStateBits.bAdditionalLink
        Rectangle (2,364 85x18), "Port A", colour toggle: g_stHMI_EL1008EcSlaveStateBits.bPortA
        Rectangle (2,384 85x18), "Port B", colour toggle: g_stHMI_EL1008EcSlaveStateBits.bPortB
        Rectangle (2,404 85x18), "Port C", colour toggle: g_stHMI_EL1008EcSlaveStateBits.bPortC
        Rectangle (2,424 85x18), "Port D", colour toggle: g_stHMI_EL1008EcSlaveStateBits.bPortD
    Group (447,42 89x451)
        RoundedRectangle (0,2 89x449)
        Label (2,0 85x25), "EL2008"
        Rectangle (2,19 85x22), "Sftw Rev: %s", text variable: g_iHMI_ProdCodeEL2008
        Rectangle (2,39 85x22), "Port A CRC: %s", text variable: g_stHMI_EL2008CrcErrorEx.portA
        Rectangle (2,59 85x22), "Port B CRC: %s", text variable: g_stHMI_EL2008CrcErrorEx.portB
        Rectangle (2,79 85x22), "Port C CRC: %s", text variable: g_stHMI_EL2008CrcErrorEx.portC
        Rectangle (2,99 85x22), "Port D CRC: %s", text variable: g_stHMI_EL2008CrcErrorEx.portD
        Rectangle (2,124 85x18), "BootStrap", colour toggle: g_stHMI_EL2008EcSlaveStateBits.bBootStrap
        Rectangle (2,144 85x18), "Init", colour toggle: g_stHMI_EL2008EcSlaveStateBits.bInit
        Rectangle (2,164 85x18), "PreOP", colour toggle: g_stHMI_EL2008EcSlaveStateBits.bPreop
        Rectangle (2,184 85x18), "SafeOP", colour toggle: g_stHMI_EL2008EcSlaveStateBits.bSafeOp
        Rectangle (2,204 85x18), "OP", colour toggle: g_stHMI_EL2008EcSlaveStateBits.bOp
        Rectangle (2,224 85x18), "Error", colour toggle: g_stHMI_EL2008EcSlaveStateBits.bError
        Rectangle (2,244 85x18), "InvVPRS", colour toggle: g_stHMI_EL2008EcSlaveStateBits.bInvVPRS
        Rectangle (2,264 85x18), "InitCmdError", colour toggle: g_stHMI_EL2008EcSlaveStateBits.bInitCmdError
        Rectangle (2,284 85x18), "LinkNotPresent", colour toggle: g_stHMI_EL2008EcSlaveStateBits.bLinkNotPresent
        Rectangle (2,304 85x18), "Link_w/o_Com", colour toggle: g_stHMI_EL2008EcSlaveStateBits.bLinkWithoutComm
        Rectangle (2,324 85x18), "LinkMissing", colour toggle: g_stHMI_EL2008EcSlaveStateBits.bLinkMissing
        Rectangle (2,344 85x18), "AdditionalLink", colour toggle: g_stHMI_EL2008EcSlaveStateBits.bAdditionalLink
        Rectangle (2,364 85x18), "Port A", colour toggle: g_stHMI_EL2008EcSlaveStateBits.bPortA
        Rectangle (2,384 85x18), "Port B", colour toggle: g_stHMI_EL2008EcSlaveStateBits.bPortB
        Rectangle (2,404 85x18), "Port C", colour toggle: g_stHMI_EL2008EcSlaveStateBits.bPortC
        Rectangle (2,424 85x18), "Port D", colour toggle: g_stHMI_EL2008EcSlaveStateBits.bPortD
    Group (536,42 89x451)
        RoundedRectangle (0,2 89x449)
        Label (2,0 85x25), "EL3002"
        Rectangle (2,19 85x22), "Sftw Rev: %s", text variable: g_iHMI_ProdCodeEL3002
        Rectangle (2,39 85x22), "Port A CRC: %s", text variable: g_stHMI_EL3002CrcErrorEx.portA
        Rectangle (2,59 85x22), "Port B CRC: %s", text variable: g_stHMI_EL3002CrcErrorEx.portB
        Rectangle (2,79 85x22), "Port C CRC: %s", text variable: g_stHMI_EL3002CrcErrorEx.portC
        Rectangle (2,99 85x22), "Port D CRC: %s", text variable: g_stHMI_EL3002CrcErrorEx.portD
        Rectangle (2,124 85x18), "BootStrap", colour toggle: g_stHMI_EL3002EcSlaveStateBits.bBootStrap
        Rectangle (2,144 85x18), "Init", colour toggle: g_stHMI_EL3002EcSlaveStateBits.bInit
        Rectangle (2,164 85x18), "PreOP", colour toggle: g_stHMI_EL3002EcSlaveStateBits.bPreop
        Rectangle (2,184 85x18), "SafeOP", colour toggle: g_stHMI_EL3002EcSlaveStateBits.bSafeOp
        Rectangle (2,204 85x18), "OP", colour toggle: g_stHMI_EL3002EcSlaveStateBits.bOp
        Rectangle (2,224 85x18), "Error", colour toggle: g_stHMI_EL3002EcSlaveStateBits.bError
        Rectangle (2,244 85x18), "InvVPRS", colour toggle: g_stHMI_EL3002EcSlaveStateBits.bInvVPRS
        Rectangle (2,264 85x18), "InitCmdError", colour toggle: g_stHMI_EL3002EcSlaveStateBits.bInitCmdError
        Rectangle (2,284 85x18), "LinkNotPresent", colour toggle: g_stHMI_EL3002EcSlaveStateBits.bLinkNotPresent
        Rectangle (2,304 85x18), "Link_w/o_Com", colour toggle: g_stHMI_EL3002EcSlaveStateBits.bLinkWithoutComm
        Rectangle (2,324 85x18), "LinkMissing", colour toggle: g_stHMI_EL3002EcSlaveStateBits.bLinkMissing
        Rectangle (2,344 85x18), "AdditionalLink", colour toggle: g_stHMI_EL3002EcSlaveStateBits.bAdditionalLink
        Rectangle (2,364 85x18), "Port A", colour toggle: g_stHMI_EL3002EcSlaveStateBits.bPortA
        Rectangle (2,384 85x18), "Port B", colour toggle: g_stHMI_EL3002EcSlaveStateBits.bPortB
        Rectangle (2,404 85x18), "Port C", colour toggle: g_stHMI_EL3002EcSlaveStateBits.bPortC
        Rectangle (2,424 85x18), "Port D", colour toggle: g_stHMI_EL3002EcSlaveStateBits.bPortD
    Group (625,42 89x451)
        RoundedRectangle (0,2 89x449)
        Label (2,0 85x25), "EL4034"
        Rectangle (2,19 85x22), "Sftw Rev: %s", text variable: g_iHMI_ProdCodeEL4034
        Rectangle (2,39 85x22), "Port A CRC: %s", text variable: g_stHMI_EL4034CrcErrorEx.portA
        Rectangle (2,59 85x22), "Port B CRC: %s", text variable: g_stHMI_EL4034CrcErrorEx.portB
        Rectangle (2,79 85x22), "Port C CRC: %s", text variable: g_stHMI_EL4034CrcErrorEx.portC
        Rectangle (2,99 85x22), "Port D CRC: %s", text variable: g_stHMI_EL4034CrcErrorEx.portD
        Rectangle (2,124 85x18), "BootStrap", colour toggle: g_stHMI_EL4034EcSlaveStateBits.bBootStrap
        Rectangle (2,144 85x18), "Init", colour toggle: g_stHMI_EL4034EcSlaveStateBits.bInit
        Rectangle (2,164 85x18), "PreOP", colour toggle: g_stHMI_EL4034EcSlaveStateBits.bPreop
        Rectangle (2,184 85x18), "SafeOP", colour toggle: g_stHMI_EL4034EcSlaveStateBits.bSafeOp
        Rectangle (2,204 85x18), "OP", colour toggle: g_stHMI_EL4034EcSlaveStateBits.bOp
        Rectangle (2,224 85x18), "Error", colour toggle: g_stHMI_EL4034EcSlaveStateBits.bError
        Rectangle (2,244 85x18), "InvVPRS", colour toggle: g_stHMI_EL4034EcSlaveStateBits.bInvVPRS
        Rectangle (2,264 85x18), "InitCmdError", colour toggle: g_stHMI_EL4034EcSlaveStateBits.bInitCmdError
        Rectangle (2,284 85x18), "LinkNotPresent", colour toggle: g_stHMI_EL4034EcSlaveStateBits.bLinkNotPresent
        Rectangle (2,304 85x18), "Link_w/o_Com", colour toggle: g_stHMI_EL4034EcSlaveStateBits.bLinkWithoutComm
        Rectangle (2,324 85x18), "LinkMissing", colour toggle: g_stHMI_EL4034EcSlaveStateBits.bLinkMissing
        Rectangle (2,344 85x18), "AdditionalLink", colour toggle: g_stHMI_EL4034EcSlaveStateBits.bAdditionalLink
        Rectangle (2,364 85x18), "Port A", colour toggle: g_stHMI_EL4034EcSlaveStateBits.bPortA
        Rectangle (2,384 85x18), "Port B", colour toggle: g_stHMI_EL4034EcSlaveStateBits.bPortB
        Rectangle (2,404 85x18), "Port C", colour toggle: g_stHMI_EL4034EcSlaveStateBits.bPortC
        Rectangle (2,424 85x18), "Port D", colour toggle: g_stHMI_EL4034EcSlaveStateBits.bPortD
    Group (714,42 89x451)
        RoundedRectangle (0,2 89x449)
        Label (2,0 85x25), "EL7201 #1"
        Rectangle (2,19 85x22), "Sftw Rev: %s", text variable: g_iHMI_ProdCodeEL7201_1
        Rectangle (2,39 85x22), "Port A CRC: %s", text variable: g_stHMI_EL7201_1CrcErrorEx.portA
        Rectangle (2,59 85x22), "Port B CRC: %s", text variable: g_stHMI_EL7201_1CrcErrorEx.portB
        Rectangle (2,79 85x22), "Port C CRC: %s", text variable: g_stHMI_EL7201_1CrcErrorEx.portC
        Rectangle (2,99 85x22), "Port D CRC: %s", text variable: g_stHMI_EL7201_1CrcErrorEx.portD
        Rectangle (2,124 85x18), "BootStrap", colour toggle: g_stHMI_EL7201_1EcSlaveStateBits.bBootStrap
        Rectangle (2,144 85x18), "Init", colour toggle: g_stHMI_EL7201_1EcSlaveStateBits.bInit
        Rectangle (2,164 85x18), "PreOP", colour toggle: g_stHMI_EL7201_1EcSlaveStateBits.bPreop
        Rectangle (2,184 85x18), "SafeOP", colour toggle: g_stHMI_EL7201_1EcSlaveStateBits.bSafeOp
        Rectangle (2,204 85x18), "OP", colour toggle: g_stHMI_EL7201_1EcSlaveStateBits.bOp
        Rectangle (2,224 85x18), "Error", colour toggle: g_stHMI_EL7201_1EcSlaveStateBits.bError
        Rectangle (2,244 85x18), "InvVPRS", colour toggle: g_stHMI_EL7201_1EcSlaveStateBits.bInvVPRS
        Rectangle (2,264 85x18), "InitCmdError", colour toggle: g_stHMI_EL7201_1EcSlaveStateBits.bInitCmdError
        Rectangle (2,284 85x18), "LinkNotPresent", colour toggle: g_stHMI_EL7201_1EcSlaveStateBits.bLinkNotPresent
        Rectangle (2,304 85x18), "Link_w/o_Com", colour toggle: g_stHMI_EL7201_1EcSlaveStateBits.bLinkWithoutComm
        Rectangle (2,324 85x18), "LinkMissing", colour toggle: g_stHMI_EL7201_1EcSlaveStateBits.bLinkMissing
        Rectangle (2,344 85x18), "AdditionalLink", colour toggle: g_stHMI_EL7201_1EcSlaveStateBits.bAdditionalLink
        Rectangle (2,364 85x18), "Port A", colour toggle: g_stHMI_EL7201_1EcSlaveStateBits.bPortA
        Rectangle (2,384 85x18), "Port B", colour toggle: g_stHMI_EL7201_1EcSlaveStateBits.bPortB
        Rectangle (2,404 85x18), "Port C", colour toggle: g_stHMI_EL7201_1EcSlaveStateBits.bPortC
        Rectangle (2,424 85x18), "Port D", colour toggle: g_stHMI_EL7201_1EcSlaveStateBits.bPortD
    Group (803,42 89x451)
        RoundedRectangle (0,2 89x449)
        Label (2,0 85x25), "EL7201 #2"
        Rectangle (2,19 85x22), "Sftw Rev: %s", text variable: g_iHMI_ProdCodeEL7201_2
        Rectangle (2,39 85x22), "Port A CRC: %s", text variable: g_stHMI_EL7201_2CrcErrorEx.portA
        Rectangle (2,59 85x22), "Port B CRC: %s", text variable: g_stHMI_EL7201_2CrcErrorEx.portB
        Rectangle (2,79 85x22), "Port C CRC: %s", text variable: g_stHMI_EL7201_2CrcErrorEx.portC
        Rectangle (2,99 85x22), "Port D CRC: %s", text variable: g_stHMI_EL7201_2CrcErrorEx.portD
        Rectangle (2,124 85x18), "BootStrap", colour toggle: g_stHMI_EL7201_2EcSlaveStateBits.bBootStrap
        Rectangle (2,144 85x18), "Init", colour toggle: g_stHMI_EL7201_2EcSlaveStateBits.bInit
        Rectangle (2,164 85x18), "PreOP", colour toggle: g_stHMI_EL7201_2EcSlaveStateBits.bPreop
        Rectangle (2,184 85x18), "SafeOP", colour toggle: g_stHMI_EL7201_2EcSlaveStateBits.bSafeOp
        Rectangle (2,204 85x18), "OP", colour toggle: g_stHMI_EL7201_2EcSlaveStateBits.bOp
        Rectangle (2,224 85x18), "Error", colour toggle: g_stHMI_EL7201_2EcSlaveStateBits.bError
        Rectangle (2,244 85x18), "InvVPRS", colour toggle: g_stHMI_EL7201_2EcSlaveStateBits.bInvVPRS
        Rectangle (2,264 85x18), "InitCmdError", colour toggle: g_stHMI_EL7201_2EcSlaveStateBits.bInitCmdError
        Rectangle (2,284 85x18), "LinkNotPresent", colour toggle: g_stHMI_EL7201_2EcSlaveStateBits.bLinkNotPresent
        Rectangle (2,304 85x18), "Link_w/o_Com", colour toggle: g_stHMI_EL7201_2EcSlaveStateBits.bLinkWithoutComm
        Rectangle (2,324 85x18), "LinkMissing", colour toggle: g_stHMI_EL7201_2EcSlaveStateBits.bLinkMissing
        Rectangle (2,344 85x18), "AdditionalLink", colour toggle: g_stHMI_EL7201_2EcSlaveStateBits.bAdditionalLink
        Rectangle (2,364 85x18), "Port A", colour toggle: g_stHMI_EL7201_2EcSlaveStateBits.bPortA
        Rectangle (2,384 85x18), "Port B", colour toggle: g_stHMI_EL7201_2EcSlaveStateBits.bPortB
        Rectangle (2,404 85x18), "Port C", colour toggle: g_stHMI_EL7201_2EcSlaveStateBits.bPortC
        Rectangle (2,424 85x18), "Port D", colour toggle: g_stHMI_EL7201_2EcSlaveStateBits.bPortD
END_VISUALIZATION

// ---- VISUs/TwinCAT_INFO.TcVIS
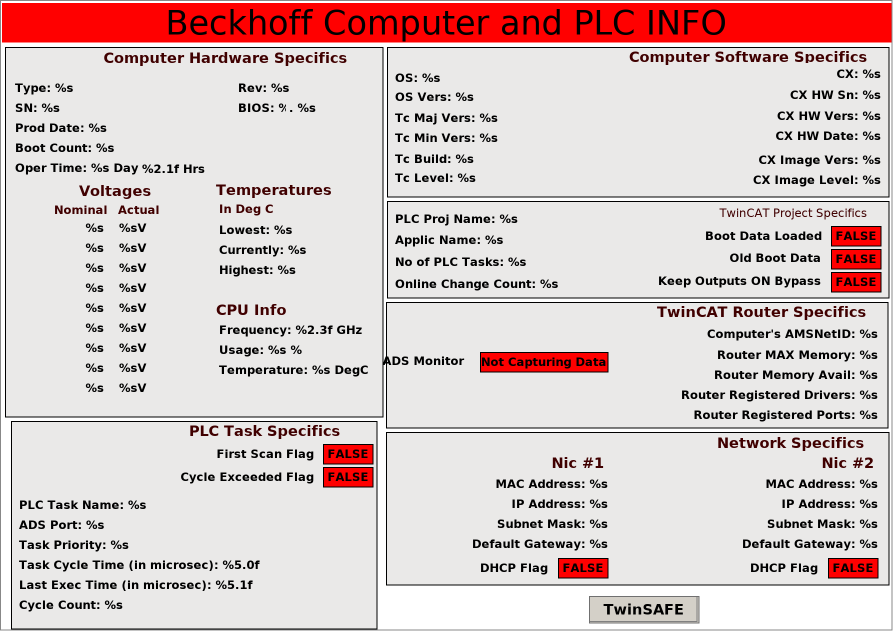
VISUALIZATION TwinCAT_INFO  // 893x631
    Button (589,596 110x27), "TwinSAFE"
        OnMouseClick: change screen: TwinSAFE
    RoundedRectangle (2,3 889x39), "Beckhoff Computer and PLC INFO"
    RoundedRectangle (387,47 502x150)
    Label (614,44 256x26), "Computer Software Specifics"
    Rectangle (392,67 256x22), "OS: %s", text variable: g_stHMI_DevIdent.strImageOsName
    RoundedRectangle (387,201 502x97)
    Label (695,200 175x26), "TwinCAT Project Specifics"
    RoundedRectangle (386,302 502x126)
    Label (613,299 256x26), "TwinCAT Router Specifics"
    RoundedRectangle (11,421 366x208)
    Label (185,418 158x26), "PLC Task Specifics"
    Rectangle (392,86 208x22), "OS Vers: %s", text variable: g_stHMI_DevIdent.strImageOsVersion
    Rectangle (392,107 119x22), "Tc Maj Vers: %s", text variable: g_stHMI_DevIdent.strTwinCATVersion
    Rectangle (392,127 111x22), "Tc Min Vers: %s", text variable: g_stHMI_DevIdent.strTwinCATRevision
    Rectangle (392,148 111x22), "Tc Build: %s", text variable: g_stHMI_DevIdent.strTwinCATBuild
    Rectangle (392,167 111x22), "Tc Level: %s", text variable: g_stHMI_DevIdent.strTwinCATLevel
    Rectangle (738,63 146x22), "CX: %s", text variable: g_stHMI_DevIdent.strHardwareModel
    Rectangle (726,84 158x22), "CX HW Sn: %s", text variable: g_stHMI_DevIdent.strHardwareSerialNo
    Rectangle (733,105 151x22), "CX HW Vers: %s", text variable: g_stHMI_DevIdent.strHardwareVersion
    Rectangle (737,125 147x22), "CX HW Date: %s", text variable: g_stHMI_DevIdent.strHardwareDate
    Rectangle (725,149 159x22), "CX Image Vers: %s", text variable: g_stHMI_DevIdent.strImageVersion
    Rectangle (625,169 259x22), "CX Image Level: %s", text variable: g_stHMI_DevIdent.strImageLevel
    Rectangle (392,208 283x22), "PLC Proj Name: %s", text variable: g_stHMI_AppInfo.ProjectName
    Rectangle (392,229 359x22), "Applic Name: %s", text variable: g_stHMI_AppInfo.AppName
    Rectangle (392,251 155x22), "No of PLC Tasks: %s", text variable: g_stHMI_AppInfo.TaskCnt
    Rectangle (392,273 191x22), "Online Change Count: %s", text variable: g_stHMI_AppInfo.OnlineChangeCnt
    Group (831,226 50x20)
        Rectangle (0,0 50x20), "TRUE", invisible if: NOT g_stHMI_AppInfo.BootDataLoaded
        Rectangle (0,0 50x20), "FALSE", invisible if: g_stHMI_AppInfo.BootDataLoaded
    Label (705,224 120x24), "Boot Data Loaded"
    Group (831,249 50x20)
        Rectangle (0,0 50x20), "TRUE", invisible if: NOT g_stHMI_AppInfo.OldBootData
        Rectangle (0,0 50x20), "FALSE", invisible if: g_stHMI_AppInfo.OldBootData
    Label (726,246 98x24), "Old Boot Data"
    Group (831,272 50x20)
        Rectangle (0,0 50x20), "TRUE", invisible if: NOT g_stHMI_AppInfo.KeepOutputsOnBP
        Rectangle (0,0 50x20), "FALSE", invisible if: NOT g_stHMI_AppInfo.KeepOutputsOnBP
    Label (682,269 142x24), "Keep Outputs ON Bypass"
    Label (392,349 75x24), "ADS Monitor"
    Group (480,352 128x20)
        Rectangle (0,0 128x20), "Capturing Data", invisible if: NOT g_stHMI_RouterStatusInfo.amsDebugLog
        Rectangle (0,0 128x20), "Not Capturing Data", invisible if: g_stHMI_RouterStatusInfo.amsDebugLog
    Rectangle (560,323 321x22), "Computer's AMSNetID: %s", text variable: g_stHMI_DevIdent.strAmsNetId
    Rectangle (673,344 208x22), "Router MAX Memory: %s", text variable: g_stHMI_RouterStatusInfo.maxMem
    Rectangle (673,364 208x22), "Router Memory Avail: %s", text variable: g_stHMI_RouterStatusInfo.maxMemAvail
    Rectangle (673,384 208x22), "Router Registered Drivers: %s", text variable: g_stHMI_RouterStatusInfo.regDrivers
    Rectangle (673,404 208x22), "Router Registered Ports: %s", text variable: g_stHMI_RouterStatusInfo.regPorts
    RoundedRectangle (5,47 378x370)
    Label (94,45 256x26), "Computer Hardware Specifics"
    Rectangle (12,77 141x22), "Type: %s", text variable: g_sHMI_MainboardType
    Rectangle (12,97 171x22), "SN: %s", text variable: g_sHMI_MainboardSN
    Rectangle (12,117 207x22), "Prod Date: %s", text variable: g_sHMI_MainboardProdDate
    Rectangle (12,137 151x22), "Boot Count: %s", text variable: g_udiHMI_MainboardBootCount
    Rectangle (12,157 184x22), "Oper Time: %s Days", text variable: g_udiHMI_MainboardOperTimeDays
    Rectangle (139,158 70x22), "%2.1f Hrs", text variable: g_lrHMI_MainboardOperTimeHrs
    Label (213,177 120x26), "Temperatures"
    Rectangle (216,219 102x22), "Lowest: %s", text variable: g_diHMI_MainboardMinTemp
    Rectangle (216,239 102x22), "Currently: %s", text variable: g_iHMI_MainboardActualTemp
    Rectangle (216,259 102x22), "Highest: %s", text variable: g_diHMI_MainboardMaxTemp
    Rectangle (235,77 67x22), "Rev: %s", text variable: g_bHMI_MainboardRevision
    Rectangle (235,97 67x22), "BIOS: %s", text variable: g_bHMI_MainboardBiosMajVers
    Rectangle (286,97 67x22), ". %s", text variable: g_bHMI_MainboardBiosMinVers
    Label (51,197 76x26), "Nominal"
    Rectangle (37,217 70x22), "%s", text variable: g_sHMI_Mainboard1p05v
    Rectangle (37,237 70x22), "%s", text variable: g_sHMI_MainboardVccCore
    Rectangle (37,257 70x22), "%s", text variable: g_sHMI_Mainboard5v
    Rectangle (37,277 70x22), "%s", text variable: g_sHMI_Mainboard12v
    Rectangle (37,297 70x22), "%s", text variable: g_sHMI_MainboardVBatt
    Rectangle (16,317 91x22), "%s", text variable: g_sHMI_MainboardPwrCtrlVcc
    Rectangle (16,337 91x22), "%s", text variable: g_sHMI_MainboardCX2100_5v
    Rectangle (18,357 89x22), "%s", text variable: g_sHMI_MainboardCX2100_12v
    Rectangle (19,377 88x22), "%s", text variable: g_sHMI_MainboardCX2100_24v
    Label (115,197 76x26), "Actual"
    Rectangle (116,217 70x22), "%sV", text variable: g_lrHMI_Mainboard1p05v
    Rectangle (116,237 70x22), "%sV", text variable: g_lrHMI_MainboardVccCore
    Rectangle (116,257 70x22), "%sV", text variable: g_lrHMI_Mainboard5v
    Rectangle (116,277 70x22), "%sV", text variable: g_lrHMI_Mainboard12v
    Rectangle (116,297 70x22), "%sV", text variable: g_lrHMI_MainboardVBatt
    Rectangle (116,317 91x22), "%sV", text variable: g_lrHMI_MainboardPwrCtrlVcc
    Rectangle (116,337 91x22), "%sV", text variable: g_lrHMI_MainboardCX2100_5v
    Rectangle (116,357 89x22), "%sV", text variable: g_lrHMI_MainboardCX2100_12v
    Rectangle (116,377 88x22), "%sV", text variable: g_lrHMI_MainboardCX2100_24v
    Label (76,178 71x26), "Voltages"
    Label (216,196 120x26), "In Deg C"
    Group (323,444 50x20)
        Rectangle (0,0 50x20), "TRUE", invisible if: NOT g_stHMI_PlcTaskSystemInfo.FirstCycle
        Rectangle (0,0 50x20), "FALSE", invisible if: g_stHMI_PlcTaskSystemInfo.FirstCycle
    Label (197,442 120x24), "First Scan Flag"
    Group (323,467 50x20)
        Rectangle (0,0 50x20), "TRUE", invisible if: NOT g_stHMI_PlcTaskSystemInfo.CycleTimeExceeded
        Rectangle (0,0 50x20), "FALSE", invisible if: g_stHMI_PlcTaskSystemInfo.CycleTimeExceeded
    Label (197,465 120x24), "Cycle Exceeded Flag"
    Rectangle (16,494 357x22), "PLC Task Name: %s", text variable: g_stHMI_PlcTaskSystemInfo.TaskName
    Rectangle (16,514 299x22), "ADS Port: %s", text variable: g_stHMI_PlcTaskSystemInfo.AdsPort
    Rectangle (16,534 214x22), "Task Priority: %s", text variable: g_stHMI_PlcTaskSystemInfo.Priority
    Rectangle (16,554 298x22), "Task Cycle Time (in microsec): %5.0f", text variable: g_lrHMI_PlcTaskSystemInfo_CycleTime
    Rectangle (16,574 298x22), "Last Exec Time (in microsec): %5.1f", text variable: g_lrHMI_PlcTaskSystemInfo_LastExecTime
    Rectangle (16,594 214x22), "Cycle Count: %s", text variable: g_stHMI_PlcTaskSystemInfo.CycleCount
    Label (213,297 120x26), "CPU Info"
    Rectangle (216,319 163x22), "Frequency: %2.3f GHz", text variable: g_lrHMI_CPUfrequency
    Rectangle (216,339 122x22), "Usage: %s %", text variable: g_iHMI_CPUusage
    Rectangle (216,359 156x22), "Temperature: %s DegC", text variable: g_iHMI_CPUtemperature
    RoundedRectangle (386,432 503x153)
    Label (716,430 151x26), "Network Specifics"
    Rectangle (396,473 215x22), "MAC Address: %s", text variable: System_Functions.ST_NIC0_ModContent.sMACAddress
    Rectangle (398,493 213x22), "IP Address: %s", text variable: System_Functions.ST_NIC0_ModContent.sIPAddress
    Rectangle (400,513 211x22), "Subnet Mask: %s", text variable: System_Functions.ST_NIC0_ModContent.sSubnetMask
    Rectangle (403,533 208x22), "Default Gateway: %s", text variable: System_Functions.ST_NIC0_ModContent.sDefaultGateway
    Group (558,558 50x20)
        Rectangle (0,0 50x20), "TRUE", invisible if: NOT System_Functions.ST_NIC0_ModContent.xDHCP
        Rectangle (0,0 50x20), "FALSE", invisible if: System_Functions.ST_NIC0_ModContent.xDHCP
    Label (481,556 70x24), "DHCP Flag"
    Label (456,450 151x26), "Nic #1"
    Rectangle (666,473 215x22), "MAC Address: %s", text variable: System_Functions.ST_NIC1_ModContent.sMACAddress
    Rectangle (668,493 213x22), "IP Address: %s", text variable: System_Functions.ST_NIC1_ModContent.sIPAddress
    Rectangle (670,513 211x22), "Subnet Mask: %s", text variable: System_Functions.ST_NIC1_ModContent.sSubnetMask
    Rectangle (673,533 208x22), "Default Gateway: %s", text variable: System_Functions.ST_NIC1_ModContent.sDefaultGateway
    Group (828,558 50x20)
        Rectangle (0,0 50x20), "TRUE", invisible if: NOT System_Functions.ST_NIC1_ModContent.xDHCP
        Rectangle (0,0 50x20), "FALSE", invisible if: System_Functions.ST_NIC1_ModContent.xDHCP
    Label (751,556 70x24), "DHCP Flag"
    Label (726,450 151x26), "Nic #2"
END_VISUALIZATION

// ---- VISUs/TwinCAT_INFO.TcVIS
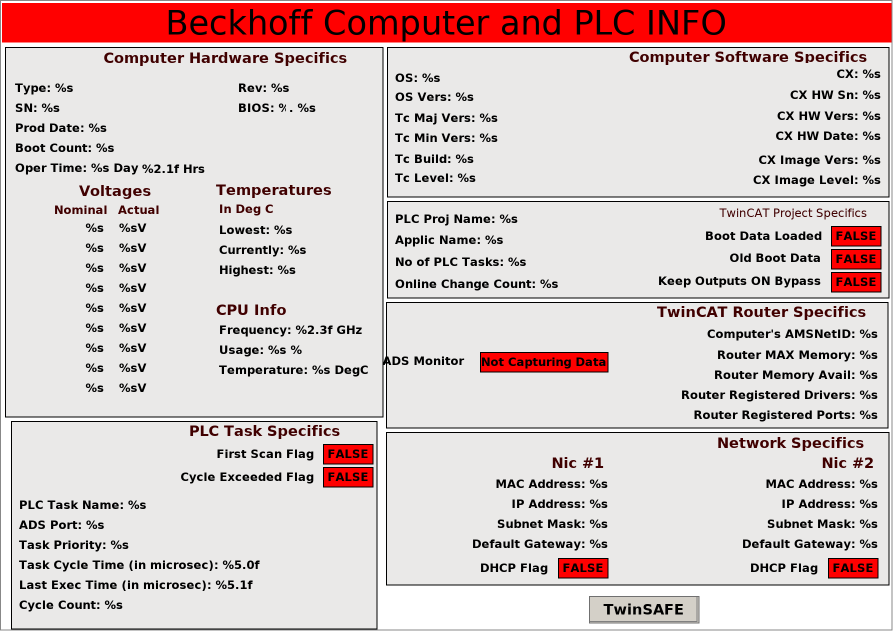
VISUALIZATION TwinCAT_INFO  // 893x631
    Button (589,596 110x27), "TwinSAFE"
        OnMouseClick: change screen: TwinSAFE
    RoundedRectangle (2,3 889x39), "Beckhoff Computer and PLC INFO"
    RoundedRectangle (387,47 502x150)
    Label (614,44 256x26), "Computer Software Specifics"
    Rectangle (392,67 256x22), "OS: %s", text variable: g_stHMI_DevIdent.strImageOsName
    RoundedRectangle (387,201 502x97)
    Label (695,200 175x26), "TwinCAT Project Specifics"
    RoundedRectangle (386,302 502x126)
    Label (613,299 256x26), "TwinCAT Router Specifics"
    RoundedRectangle (11,421 366x208)
    Label (185,418 158x26), "PLC Task Specifics"
    Rectangle (392,86 208x22), "OS Vers: %s", text variable: g_stHMI_DevIdent.strImageOsVersion
    Rectangle (392,107 119x22), "Tc Maj Vers: %s", text variable: g_stHMI_DevIdent.strTwinCATVersion
    Rectangle (392,127 111x22), "Tc Min Vers: %s", text variable: g_stHMI_DevIdent.strTwinCATRevision
    Rectangle (392,148 111x22), "Tc Build: %s", text variable: g_stHMI_DevIdent.strTwinCATBuild
    Rectangle (392,167 111x22), "Tc Level: %s", text variable: g_stHMI_DevIdent.strTwinCATLevel
    Rectangle (738,63 146x22), "CX: %s", text variable: g_stHMI_DevIdent.strHardwareModel
    Rectangle (726,84 158x22), "CX HW Sn: %s", text variable: g_stHMI_DevIdent.strHardwareSerialNo
    Rectangle (733,105 151x22), "CX HW Vers: %s", text variable: g_stHMI_DevIdent.strHardwareVersion
    Rectangle (737,125 147x22), "CX HW Date: %s", text variable: g_stHMI_DevIdent.strHardwareDate
    Rectangle (725,149 159x22), "CX Image Vers: %s", text variable: g_stHMI_DevIdent.strImageVersion
    Rectangle (625,169 259x22), "CX Image Level: %s", text variable: g_stHMI_DevIdent.strImageLevel
    Rectangle (392,208 283x22), "PLC Proj Name: %s", text variable: g_stHMI_AppInfo.ProjectName
    Rectangle (392,229 359x22), "Applic Name: %s", text variable: g_stHMI_AppInfo.AppName
    Rectangle (392,251 155x22), "No of PLC Tasks: %s", text variable: g_stHMI_AppInfo.TaskCnt
    Rectangle (392,273 191x22), "Online Change Count: %s", text variable: g_stHMI_AppInfo.OnlineChangeCnt
    Group (831,226 50x20)
        Rectangle (0,0 50x20), "TRUE", invisible if: NOT g_stHMI_AppInfo.BootDataLoaded
        Rectangle (0,0 50x20), "FALSE", invisible if: g_stHMI_AppInfo.BootDataLoaded
    Label (705,224 120x24), "Boot Data Loaded"
    Group (831,249 50x20)
        Rectangle (0,0 50x20), "TRUE", invisible if: NOT g_stHMI_AppInfo.OldBootData
        Rectangle (0,0 50x20), "FALSE", invisible if: g_stHMI_AppInfo.OldBootData
    Label (726,246 98x24), "Old Boot Data"
    Group (831,272 50x20)
        Rectangle (0,0 50x20), "TRUE", invisible if: NOT g_stHMI_AppInfo.KeepOutputsOnBP
        Rectangle (0,0 50x20), "FALSE", invisible if: NOT g_stHMI_AppInfo.KeepOutputsOnBP
    Label (682,269 142x24), "Keep Outputs ON Bypass"
    Label (392,349 75x24), "ADS Monitor"
    Group (480,352 128x20)
        Rectangle (0,0 128x20), "Capturing Data", invisible if: NOT g_stHMI_RouterStatusInfo.amsDebugLog
        Rectangle (0,0 128x20), "Not Capturing Data", invisible if: g_stHMI_RouterStatusInfo.amsDebugLog
    Rectangle (560,323 321x22), "Computer's AMSNetID: %s", text variable: g_stHMI_DevIdent.strAmsNetId
    Rectangle (673,344 208x22), "Router MAX Memory: %s", text variable: g_stHMI_RouterStatusInfo.maxMem
    Rectangle (673,364 208x22), "Router Memory Avail: %s", text variable: g_stHMI_RouterStatusInfo.maxMemAvail
    Rectangle (673,384 208x22), "Router Registered Drivers: %s", text variable: g_stHMI_RouterStatusInfo.regDrivers
    Rectangle (673,404 208x22), "Router Registered Ports: %s", text variable: g_stHMI_RouterStatusInfo.regPorts
    RoundedRectangle (5,47 378x370)
    Label (94,45 256x26), "Computer Hardware Specifics"
    Rectangle (12,77 141x22), "Type: %s", text variable: g_sHMI_MainboardType
    Rectangle (12,97 171x22), "SN: %s", text variable: g_sHMI_MainboardSN
    Rectangle (12,117 207x22), "Prod Date: %s", text variable: g_sHMI_MainboardProdDate
    Rectangle (12,137 151x22), "Boot Count: %s", text variable: g_udiHMI_MainboardBootCount
    Rectangle (12,157 184x22), "Oper Time: %s Days", text variable: g_udiHMI_MainboardOperTimeDays
    Rectangle (139,158 70x22), "%2.1f Hrs", text variable: g_lrHMI_MainboardOperTimeHrs
    Label (213,177 120x26), "Temperatures"
    Rectangle (216,219 102x22), "Lowest: %s", text variable: g_diHMI_MainboardMinTemp
    Rectangle (216,239 102x22), "Currently: %s", text variable: g_iHMI_MainboardActualTemp
    Rectangle (216,259 102x22), "Highest: %s", text variable: g_diHMI_MainboardMaxTemp
    Rectangle (235,77 67x22), "Rev: %s", text variable: g_bHMI_MainboardRevision
    Rectangle (235,97 67x22), "BIOS: %s", text variable: g_bHMI_MainboardBiosMajVers
    Rectangle (286,97 67x22), ". %s", text variable: g_bHMI_MainboardBiosMinVers
    Label (51,197 76x26), "Nominal"
    Rectangle (37,217 70x22), "%s", text variable: g_sHMI_Mainboard1p05v
    Rectangle (37,237 70x22), "%s", text variable: g_sHMI_MainboardVccCore
    Rectangle (37,257 70x22), "%s", text variable: g_sHMI_Mainboard5v
    Rectangle (37,277 70x22), "%s", text variable: g_sHMI_Mainboard12v
    Rectangle (37,297 70x22), "%s", text variable: g_sHMI_MainboardVBatt
    Rectangle (16,317 91x22), "%s", text variable: g_sHMI_MainboardPwrCtrlVcc
    Rectangle (16,337 91x22), "%s", text variable: g_sHMI_MainboardCX2100_5v
    Rectangle (18,357 89x22), "%s", text variable: g_sHMI_MainboardCX2100_12v
    Rectangle (19,377 88x22), "%s", text variable: g_sHMI_MainboardCX2100_24v
    Label (115,197 76x26), "Actual"
    Rectangle (116,217 70x22), "%sV", text variable: g_lrHMI_Mainboard1p05v
    Rectangle (116,237 70x22), "%sV", text variable: g_lrHMI_MainboardVccCore
    Rectangle (116,257 70x22), "%sV", text variable: g_lrHMI_Mainboard5v
    Rectangle (116,277 70x22), "%sV", text variable: g_lrHMI_Mainboard12v
    Rectangle (116,297 70x22), "%sV", text variable: g_lrHMI_MainboardVBatt
    Rectangle (116,317 91x22), "%sV", text variable: g_lrHMI_MainboardPwrCtrlVcc
    Rectangle (116,337 91x22), "%sV", text variable: g_lrHMI_MainboardCX2100_5v
    Rectangle (116,357 89x22), "%sV", text variable: g_lrHMI_MainboardCX2100_12v
    Rectangle (116,377 88x22), "%sV", text variable: g_lrHMI_MainboardCX2100_24v
    Label (76,178 71x26), "Voltages"
    Label (216,196 120x26), "In Deg C"
    Group (323,444 50x20)
        Rectangle (0,0 50x20), "TRUE", invisible if: NOT g_stHMI_PlcTaskSystemInfo.FirstCycle
        Rectangle (0,0 50x20), "FALSE", invisible if: g_stHMI_PlcTaskSystemInfo.FirstCycle
    Label (197,442 120x24), "First Scan Flag"
    Group (323,467 50x20)
        Rectangle (0,0 50x20), "TRUE", invisible if: NOT g_stHMI_PlcTaskSystemInfo.CycleTimeExceeded
        Rectangle (0,0 50x20), "FALSE", invisible if: g_stHMI_PlcTaskSystemInfo.CycleTimeExceeded
    Label (197,465 120x24), "Cycle Exceeded Flag"
    Rectangle (16,494 357x22), "PLC Task Name: %s", text variable: g_stHMI_PlcTaskSystemInfo.TaskName
    Rectangle (16,514 299x22), "ADS Port: %s", text variable: g_stHMI_PlcTaskSystemInfo.AdsPort
    Rectangle (16,534 214x22), "Task Priority: %s", text variable: g_stHMI_PlcTaskSystemInfo.Priority
    Rectangle (16,554 298x22), "Task Cycle Time (in microsec): %5.0f", text variable: g_lrHMI_PlcTaskSystemInfo_CycleTime
    Rectangle (16,574 298x22), "Last Exec Time (in microsec): %5.1f", text variable: g_lrHMI_PlcTaskSystemInfo_LastExecTime
    Rectangle (16,594 214x22), "Cycle Count: %s", text variable: g_stHMI_PlcTaskSystemInfo.CycleCount
    Label (213,297 120x26), "CPU Info"
    Rectangle (216,319 163x22), "Frequency: %2.3f GHz", text variable: g_lrHMI_CPUfrequency
    Rectangle (216,339 122x22), "Usage: %s %", text variable: g_iHMI_CPUusage
    Rectangle (216,359 156x22), "Temperature: %s DegC", text variable: g_iHMI_CPUtemperature
    RoundedRectangle (386,432 503x153)
    Label (716,430 151x26), "Network Specifics"
    Rectangle (396,473 215x22), "MAC Address: %s", text variable: System_Functions.ST_NIC0_ModContent.sMACAddress
    Rectangle (398,493 213x22), "IP Address: %s", text variable: System_Functions.ST_NIC0_ModContent.sIPAddress
    Rectangle (400,513 211x22), "Subnet Mask: %s", text variable: System_Functions.ST_NIC0_ModContent.sSubnetMask
    Rectangle (403,533 208x22), "Default Gateway: %s", text variable: System_Functions.ST_NIC0_ModContent.sDefaultGateway
    Group (558,558 50x20)
        Rectangle (0,0 50x20), "TRUE", invisible if: NOT System_Functions.ST_NIC0_ModContent.xDHCP
        Rectangle (0,0 50x20), "FALSE", invisible if: System_Functions.ST_NIC0_ModContent.xDHCP
    Label (481,556 70x24), "DHCP Flag"
    Label (456,450 151x26), "Nic #1"
    Rectangle (666,473 215x22), "MAC Address: %s", text variable: System_Functions.ST_NIC1_ModContent.sMACAddress
    Rectangle (668,493 213x22), "IP Address: %s", text variable: System_Functions.ST_NIC1_ModContent.sIPAddress
    Rectangle (670,513 211x22), "Subnet Mask: %s", text variable: System_Functions.ST_NIC1_ModContent.sSubnetMask
    Rectangle (673,533 208x22), "Default Gateway: %s", text variable: System_Functions.ST_NIC1_ModContent.sDefaultGateway
    Group (828,558 50x20)
        Rectangle (0,0 50x20), "TRUE", invisible if: NOT System_Functions.ST_NIC1_ModContent.xDHCP
        Rectangle (0,0 50x20), "FALSE", invisible if: System_Functions.ST_NIC1_ModContent.xDHCP
    Label (751,556 70x24), "DHCP Flag"
    Label (726,450 151x26), "Nic #2"
END_VISUALIZATION

// ---- VISUs/TwinCAT_INFO.TcVIS
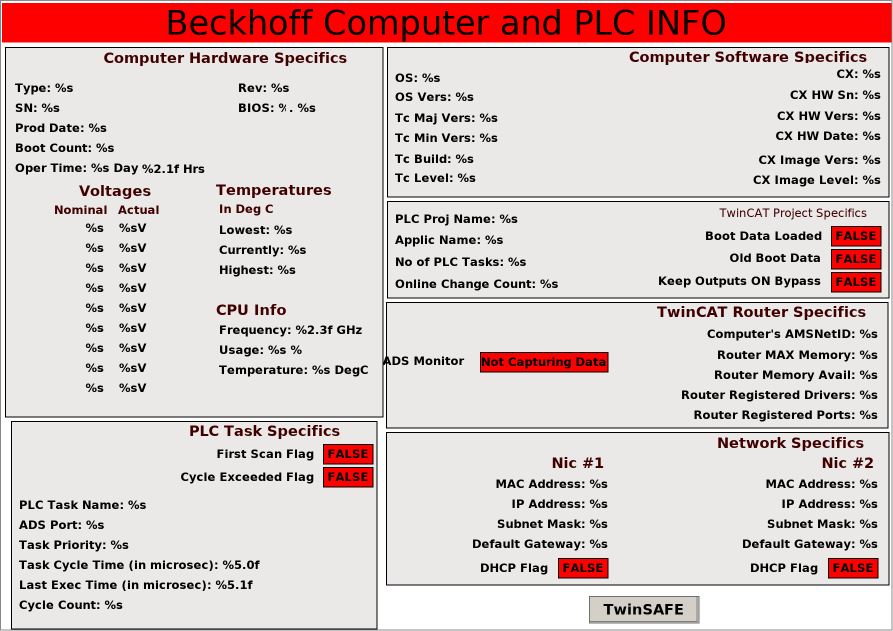
VISUALIZATION TwinCAT_INFO  // 893x631
    Button (589,596 110x27), "TwinSAFE"
        OnMouseClick: change screen: TwinSAFE
    RoundedRectangle (2,3 889x39), "Beckhoff Computer and PLC INFO"
    RoundedRectangle (387,47 502x150)
    Label (614,44 256x26), "Computer Software Specifics"
    Rectangle (392,67 256x22), "OS: %s", text variable: g_stHMI_DevIdent.strImageOsName
    RoundedRectangle (387,201 502x97)
    Label (695,200 175x26), "TwinCAT Project Specifics"
    RoundedRectangle (386,302 502x126)
    Label (613,299 256x26), "TwinCAT Router Specifics"
    RoundedRectangle (11,421 366x208)
    Label (185,418 158x26), "PLC Task Specifics"
    Rectangle (392,86 208x22), "OS Vers: %s", text variable: g_stHMI_DevIdent.strImageOsVersion
    Rectangle (392,107 119x22), "Tc Maj Vers: %s", text variable: g_stHMI_DevIdent.strTwinCATVersion
    Rectangle (392,127 111x22), "Tc Min Vers: %s", text variable: g_stHMI_DevIdent.strTwinCATRevision
    Rectangle (392,148 111x22), "Tc Build: %s", text variable: g_stHMI_DevIdent.strTwinCATBuild
    Rectangle (392,167 111x22), "Tc Level: %s", text variable: g_stHMI_DevIdent.strTwinCATLevel
    Rectangle (738,63 146x22), "CX: %s", text variable: g_stHMI_DevIdent.strHardwareModel
    Rectangle (726,84 158x22), "CX HW Sn: %s", text variable: g_stHMI_DevIdent.strHardwareSerialNo
    Rectangle (733,105 151x22), "CX HW Vers: %s", text variable: g_stHMI_DevIdent.strHardwareVersion
    Rectangle (737,125 147x22), "CX HW Date: %s", text variable: g_stHMI_DevIdent.strHardwareDate
    Rectangle (725,149 159x22), "CX Image Vers: %s", text variable: g_stHMI_DevIdent.strImageVersion
    Rectangle (625,169 259x22), "CX Image Level: %s", text variable: g_stHMI_DevIdent.strImageLevel
    Rectangle (392,208 283x22), "PLC Proj Name: %s", text variable: g_stHMI_AppInfo.ProjectName
    Rectangle (392,229 359x22), "Applic Name: %s", text variable: g_stHMI_AppInfo.AppName
    Rectangle (392,251 155x22), "No of PLC Tasks: %s", text variable: g_stHMI_AppInfo.TaskCnt
    Rectangle (392,273 191x22), "Online Change Count: %s", text variable: g_stHMI_AppInfo.OnlineChangeCnt
    Group (831,226 50x20)
        Rectangle (0,0 50x20), "TRUE", invisible if: NOT g_stHMI_AppInfo.BootDataLoaded
        Rectangle (0,0 50x20), "FALSE", invisible if: g_stHMI_AppInfo.BootDataLoaded
    Label (705,224 120x24), "Boot Data Loaded"
    Group (831,249 50x20)
        Rectangle (0,0 50x20), "TRUE", invisible if: NOT g_stHMI_AppInfo.OldBootData
        Rectangle (0,0 50x20), "FALSE", invisible if: g_stHMI_AppInfo.OldBootData
    Label (726,246 98x24), "Old Boot Data"
    Group (831,272 50x20)
        Rectangle (0,0 50x20), "TRUE", invisible if: NOT g_stHMI_AppInfo.KeepOutputsOnBP
        Rectangle (0,0 50x20), "FALSE", invisible if: NOT g_stHMI_AppInfo.KeepOutputsOnBP
    Label (682,269 142x24), "Keep Outputs ON Bypass"
    Label (392,349 75x24), "ADS Monitor"
    Group (480,352 128x20)
        Rectangle (0,0 128x20), "Capturing Data", invisible if: NOT g_stHMI_RouterStatusInfo.amsDebugLog
        Rectangle (0,0 128x20), "Not Capturing Data", invisible if: g_stHMI_RouterStatusInfo.amsDebugLog
    Rectangle (560,323 321x22), "Computer's AMSNetID: %s", text variable: g_stHMI_DevIdent.strAmsNetId
    Rectangle (673,344 208x22), "Router MAX Memory: %s", text variable: g_stHMI_RouterStatusInfo.maxMem
    Rectangle (673,364 208x22), "Router Memory Avail: %s", text variable: g_stHMI_RouterStatusInfo.maxMemAvail
    Rectangle (673,384 208x22), "Router Registered Drivers: %s", text variable: g_stHMI_RouterStatusInfo.regDrivers
    Rectangle (673,404 208x22), "Router Registered Ports: %s", text variable: g_stHMI_RouterStatusInfo.regPorts
    RoundedRectangle (5,47 378x370)
    Label (94,45 256x26), "Computer Hardware Specifics"
    Rectangle (12,77 141x22), "Type: %s", text variable: g_sHMI_MainboardType
    Rectangle (12,97 171x22), "SN: %s", text variable: g_sHMI_MainboardSN
    Rectangle (12,117 207x22), "Prod Date: %s", text variable: g_sHMI_MainboardProdDate
    Rectangle (12,137 151x22), "Boot Count: %s", text variable: g_udiHMI_MainboardBootCount
    Rectangle (12,157 184x22), "Oper Time: %s Days", text variable: g_udiHMI_MainboardOperTimeDays
    Rectangle (139,158 70x22), "%2.1f Hrs", text variable: g_lrHMI_MainboardOperTimeHrs
    Label (213,177 120x26), "Temperatures"
    Rectangle (216,219 102x22), "Lowest: %s", text variable: g_diHMI_MainboardMinTemp
    Rectangle (216,239 102x22), "Currently: %s", text variable: g_iHMI_MainboardActualTemp
    Rectangle (216,259 102x22), "Highest: %s", text variable: g_diHMI_MainboardMaxTemp
    Rectangle (235,77 67x22), "Rev: %s", text variable: g_bHMI_MainboardRevision
    Rectangle (235,97 67x22), "BIOS: %s", text variable: g_bHMI_MainboardBiosMajVers
    Rectangle (286,97 67x22), ". %s", text variable: g_bHMI_MainboardBiosMinVers
    Label (51,197 76x26), "Nominal"
    Rectangle (37,217 70x22), "%s", text variable: g_sHMI_Mainboard1p05v
    Rectangle (37,237 70x22), "%s", text variable: g_sHMI_MainboardVccCore
    Rectangle (37,257 70x22), "%s", text variable: g_sHMI_Mainboard5v
    Rectangle (37,277 70x22), "%s", text variable: g_sHMI_Mainboard12v
    Rectangle (37,297 70x22), "%s", text variable: g_sHMI_MainboardVBatt
    Rectangle (16,317 91x22), "%s", text variable: g_sHMI_MainboardPwrCtrlVcc
    Rectangle (16,337 91x22), "%s", text variable: g_sHMI_MainboardCX2100_5v
    Rectangle (18,357 89x22), "%s", text variable: g_sHMI_MainboardCX2100_12v
    Rectangle (19,377 88x22), "%s", text variable: g_sHMI_MainboardCX2100_24v
    Label (115,197 76x26), "Actual"
    Rectangle (116,217 70x22), "%sV", text variable: g_lrHMI_Mainboard1p05v
    Rectangle (116,237 70x22), "%sV", text variable: g_lrHMI_MainboardVccCore
    Rectangle (116,257 70x22), "%sV", text variable: g_lrHMI_Mainboard5v
    Rectangle (116,277 70x22), "%sV", text variable: g_lrHMI_Mainboard12v
    Rectangle (116,297 70x22), "%sV", text variable: g_lrHMI_MainboardVBatt
    Rectangle (116,317 91x22), "%sV", text variable: g_lrHMI_MainboardPwrCtrlVcc
    Rectangle (116,337 91x22), "%sV", text variable: g_lrHMI_MainboardCX2100_5v
    Rectangle (116,357 89x22), "%sV", text variable: g_lrHMI_MainboardCX2100_12v
    Rectangle (116,377 88x22), "%sV", text variable: g_lrHMI_MainboardCX2100_24v
    Label (76,178 71x26), "Voltages"
    Label (216,196 120x26), "In Deg C"
    Group (323,444 50x20)
        Rectangle (0,0 50x20), "TRUE", invisible if: NOT g_stHMI_PlcTaskSystemInfo.FirstCycle
        Rectangle (0,0 50x20), "FALSE", invisible if: g_stHMI_PlcTaskSystemInfo.FirstCycle
    Label (197,442 120x24), "First Scan Flag"
    Group (323,467 50x20)
        Rectangle (0,0 50x20), "TRUE", invisible if: NOT g_stHMI_PlcTaskSystemInfo.CycleTimeExceeded
        Rectangle (0,0 50x20), "FALSE", invisible if: g_stHMI_PlcTaskSystemInfo.CycleTimeExceeded
    Label (197,465 120x24), "Cycle Exceeded Flag"
    Rectangle (16,494 357x22), "PLC Task Name: %s", text variable: g_stHMI_PlcTaskSystemInfo.TaskName
    Rectangle (16,514 299x22), "ADS Port: %s", text variable: g_stHMI_PlcTaskSystemInfo.AdsPort
    Rectangle (16,534 214x22), "Task Priority: %s", text variable: g_stHMI_PlcTaskSystemInfo.Priority
    Rectangle (16,554 298x22), "Task Cycle Time (in microsec): %5.0f", text variable: g_lrHMI_PlcTaskSystemInfo_CycleTime
    Rectangle (16,574 298x22), "Last Exec Time (in microsec): %5.1f", text variable: g_lrHMI_PlcTaskSystemInfo_LastExecTime
    Rectangle (16,594 214x22), "Cycle Count: %s", text variable: g_stHMI_PlcTaskSystemInfo.CycleCount
    Label (213,297 120x26), "CPU Info"
    Rectangle (216,319 163x22), "Frequency: %2.3f GHz", text variable: g_lrHMI_CPUfrequency
    Rectangle (216,339 122x22), "Usage: %s %", text variable: g_iHMI_CPUusage
    Rectangle (216,359 156x22), "Temperature: %s DegC", text variable: g_iHMI_CPUtemperature
    RoundedRectangle (386,432 503x153)
    Label (716,430 151x26), "Network Specifics"
    Rectangle (396,473 215x22), "MAC Address: %s", text variable: System_Functions.ST_NIC0_ModContent.sMACAddress
    Rectangle (398,493 213x22), "IP Address: %s", text variable: System_Functions.ST_NIC0_ModContent.sIPAddress
    Rectangle (400,513 211x22), "Subnet Mask: %s", text variable: System_Functions.ST_NIC0_ModContent.sSubnetMask
    Rectangle (403,533 208x22), "Default Gateway: %s", text variable: System_Functions.ST_NIC0_ModContent.sDefaultGateway
    Group (558,558 50x20)
        Rectangle (0,0 50x20), "TRUE", invisible if: NOT System_Functions.ST_NIC0_ModContent.xDHCP
        Rectangle (0,0 50x20), "FALSE", invisible if: System_Functions.ST_NIC0_ModContent.xDHCP
    Label (481,556 70x24), "DHCP Flag"
    Label (456,450 151x26), "Nic #1"
    Rectangle (666,473 215x22), "MAC Address: %s", text variable: System_Functions.ST_NIC1_ModContent.sMACAddress
    Rectangle (668,493 213x22), "IP Address: %s", text variable: System_Functions.ST_NIC1_ModContent.sIPAddress
    Rectangle (670,513 211x22), "Subnet Mask: %s", text variable: System_Functions.ST_NIC1_ModContent.sSubnetMask
    Rectangle (673,533 208x22), "Default Gateway: %s", text variable: System_Functions.ST_NIC1_ModContent.sDefaultGateway
    Group (828,558 50x20)
        Rectangle (0,0 50x20), "TRUE", invisible if: NOT System_Functions.ST_NIC1_ModContent.xDHCP
        Rectangle (0,0 50x20), "FALSE", invisible if: System_Functions.ST_NIC1_ModContent.xDHCP
    Label (751,556 70x24), "DHCP Flag"
    Label (726,450 151x26), "Nic #2"
END_VISUALIZATION

// ---- VISUs/TwinSAFE.TcVIS
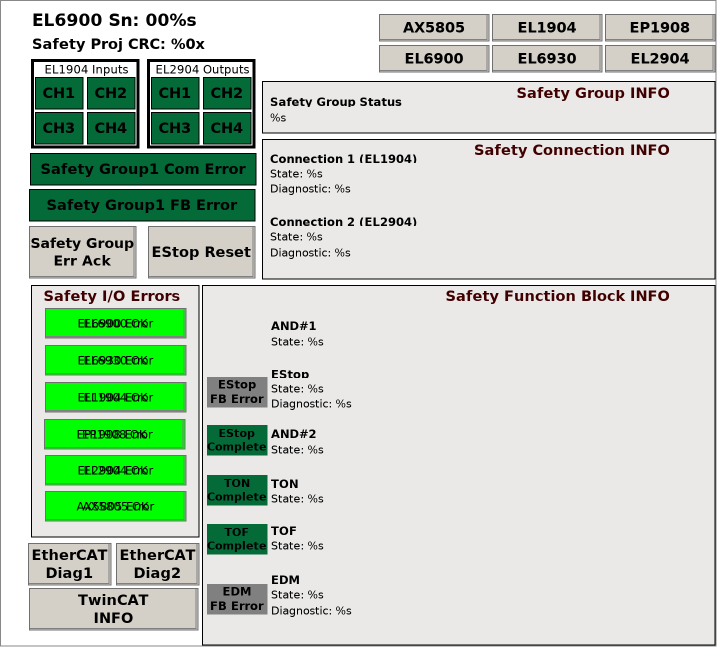
VISUALIZATION TwinSAFE  // 717x647
    RoundedRectangle (31,285 168x252)
    Rectangle (31,59 108x89)
    Rectangle (29,9 219x22), "EL6900 Sn: 00%s", text variable: g_udiHMI_SerialNumber
    Rectangle (29,33 232x22), "Safety Proj CRC: %0x", text variable: g_uiHMI_ProjectCRC
    Rectangle (35,77 48x32), "CH1", colour toggle: g_xHMI_EL1904Ch1
    Rectangle (87,77 48x32), "CH2", colour toggle: g_xHMI_EL1904Ch2
    Rectangle (35,112 48x32), "CH3", colour toggle: g_xHMI_EL1904Ch3
    Rectangle (87,112 48x32), "CH4", colour toggle: g_xHMI_EL1904Ch4
    Label (37,58 99x23), "EL1904 Inputs"
    Rectangle (147,59 108x89)
    Rectangle (151,77 48x32), "CH1", colour toggle: g_xHMI_EL2904Ch1
    Rectangle (203,77 48x32), "CH2", colour toggle: g_xHMI_EL2904Ch2
    Rectangle (151,112 48x32), "CH3", colour toggle: g_xHMI_EL2904Ch3
    Rectangle (203,112 48x32), "CH4", colour toggle: g_xHMI_EL2904Ch4
    Label (153,58 99x23), "EL2904 Outputs"
    Button (29,226 107x52), "Safety Group Err Ack"
        OnMouseDown: execute { g_xHMI_ErrAckPB := TRUE ; }
        OnMouseUp: execute { g_xHMI_ErrAckPB := FALSE ; }
    Button (148,226 107x52), "EStop Reset"
        OnMouseDown: execute { g_xHMI_EStopResetPB := TRUE ; }
        OnMouseUp: execute { g_xHMI_EStopResetPB := FALSE ; }
    Rectangle (30,153 226x32), "Safety Group1 Com Error", colour toggle: g_xHMI_SafetyGroup1_COMerrorLT
    Rectangle (29,189 226x32), "Safety Group1 FB Error", colour toggle: g_xHMI_SafetyGroup1_FBerrorLT
    Label (50,283 133x26), "Safety I/O Errors"
    Button (28,543 83x42), "EtherCAT Diag1"
        OnMouseClick: change screen: EtherCAT_Diag1
    Button (116,543 83x42), "EtherCAT Diag2"
        OnMouseClick: change screen: EtherCAT_Diag2
    Button (29,588 169x42), "TwinCAT INFO"
        OnMouseClick: change screen: TwinCAT_INFO
    RoundedRectangle (262,81 453x52)
    Label (449,80 224x26), "Safety Group INFO"
    Label (267,89 135x26), "Safety Group Status"
    RoundedRectangle (262,139 453x140)
    Label (449,137 224x26), "Safety Connection INFO"
    Label (267,146 203x26), "Connection 1 (EL1904)"
    Label (267,209 203x26), "Connection 2 (EL2904)"
    RoundedRectangle (202,285 513x360)
    Label (449,283 224x26), "Safety Function Block INFO"
    Label (268,313 50x26), "AND#1"
    Label (268,362 51x25), "EStop"
    Button (379,14 110x27), "AX5805"
        OnMouseClick: change screen: AX5805_Specific_Diagnostics
    Button (379,45 110x27), "EL6900"
        OnMouseClick: change screen: EL6900_Specific_Diagnostics
    Button (492,14 110x27), "EL1904"
        OnMouseClick: change screen: EL1904_Specific_Diagnostics
    Button (492,45 110x27), "EL6930"
        OnMouseClick: change screen: EL6930_Specific_Diagnostics
    Button (605,14 110x27), "EP1908"
        OnMouseClick: change screen: EP1908_Specific_Diagnostics
    Button (605,45 110x27), "EL2904"
        OnMouseClick: change screen: EL2904_Specific_Diagnostics
    Rectangle (267,107 321x22), "%s", text variable: g_sHMI_StatusGroup1
    Rectangle (267,163 321x22), "State: %s", text variable: g_sHMI_StateConn1
    Rectangle (267,178 386x22), "Diagnostic: %s", text variable: g_sHMI_DiagConn1
    Rectangle (267,226 321x22), "State: %s", text variable: g_sHMI_StateConn2
    Rectangle (267,242 389x22), "Diagnostic: %s", text variable: g_sHMI_DiagConn2
    Rectangle (268,331 439x22), "State: %s", text variable: g_sHMI_StatusAND1
    Rectangle (268,378 439x22), "State: %s", text variable: g_sHMI_StatusEStop1
    Rectangle (268,393 439x22), "Diagnostic: %s", text variable: g_sHMI_DiagEStop1
    Rectangle (268,439 439x22), "State: %s", text variable: g_sHMI_StatusAND2
    Label (268,421 54x26), "AND#2"
    Rectangle (268,488 439x22), "State: %s", text variable: g_sHMI_StatusTON
    Label (268,471 36x26), "TON"
    Rectangle (268,535 439x22), "State: %s", text variable: g_sHMI_StatusTOF
    Label (268,518 33x26), "TOF"
    Label (268,571 34x18), "EDM"
    Rectangle (268,584 439x22), "State: %s", text variable: g_sHMI_StatusEDM
    Rectangle (268,600 439x22), "Diagnostic: %s", text variable: g_sHMI_DiagEDM
    Rectangle (207,377 60x30), "EStop FB Error", colour toggle: g_xHMI_EStop_errorLT
    Rectangle (207,425 60x30), "EStop Complete", colour toggle: g_xHMI_EStop_CompleteLT
    Rectangle (207,475 60x30), "TON Complete", colour toggle: g_xHMI_EStop_ON_Delay_CompleteLT
    Rectangle (207,524 60x30), "TOF Complete", colour toggle: g_xHMI_EStop_OFF_Delay_CompleteLT
    Rectangle (207,584 60x30), "EDM FB Error", colour toggle: g_xHMI_EDMerrorLT
    Group (45,308 141x30)
        Button (0,0 141x30), colour toggle: g_xHMI_EL6900_General_Error
            OnMouseClick: change screen: AX5805_Specific_Diagnostics
            OnMouseUp: execute { g_xHMI_ErrAckPB := FALSE ; }
        Label (10,3 121x25), "EL6900 Error", invisible if: NOT g_xHMI_EL6900_General_Error
        Label (10,3 121x25), "EL6900 OK", invisible if: g_xHMI_EL6900_General_Error
    Group (45,345 141x30)
        Button (0,0 141x30), colour toggle: g_xHMI_EL6930_General_Error
            OnMouseClick: change screen: AX5805_Specific_Diagnostics
            OnMouseUp: execute { g_xHMI_ErrAckPB := FALSE ; }
        Label (10,3 121x25), "EL6930 Error", invisible if: NOT g_xHMI_EL6930_General_Error
        Label (10,3 121x25), "EL6930 OK", invisible if: g_xHMI_EL6930_General_Error
    Group (45,382 141x30)
        Button (0,0 141x30), colour toggle: g_xHMI_EL1904_General_Error
            OnMouseClick: change screen: AX5805_Specific_Diagnostics
            OnMouseUp: execute { g_xHMI_ErrAckPB := FALSE ; }
        Label (10,3 121x25), "EL1904 Error", invisible if: NOT g_xHMI_EL1904_General_Error
        Label (10,3 121x25), "EL1904 OK", invisible if: g_xHMI_EL1904_General_Error
    Group (44,419 141x30)
        Button (0,0 141x30), colour toggle: g_xHMI_EP1908_General_Error
            OnMouseClick: change screen: AX5805_Specific_Diagnostics
            OnMouseUp: execute { g_xHMI_ErrAckPB := FALSE ; }
        Label (10,3 121x25), "EP1908 Error", invisible if: NOT g_xHMI_EP1908_General_Error
        Label (10,3 121x25), "EP1908 OK", invisible if: g_xHMI_EP1908_General_Error
    Group (45,455 141x30)
        Button (0,0 141x30), colour toggle: g_xHMI_EL2904_General_Error
            OnMouseClick: change screen: AX5805_Specific_Diagnostics
            OnMouseUp: execute { g_xHMI_ErrAckPB := FALSE ; }
        Label (10,3 121x25), "EL2904 Error", invisible if: NOT g_xHMI_EL2904_General_Error
        Label (10,3 121x25), "EL2904 OK", invisible if: g_xHMI_EL2904_General_Error
    Group (45,491 141x30)
        Button (0,0 141x30), colour toggle: g_xHMI_AX5805_General_Error
            OnMouseClick: change screen: AX5805_Specific_Diagnostics
            OnMouseUp: execute { g_xHMI_ErrAckPB := FALSE ; }
        Label (10,3 121x25), "AX5805 Error", invisible if: NOT g_xHMI_AX5805_General_Error
        Label (10,3 121x25), "AX5805 OK", invisible if: g_xHMI_AX5805_General_Error
END_VISUALIZATION

// ---- VISUs/TwinSAFE.TcVIS
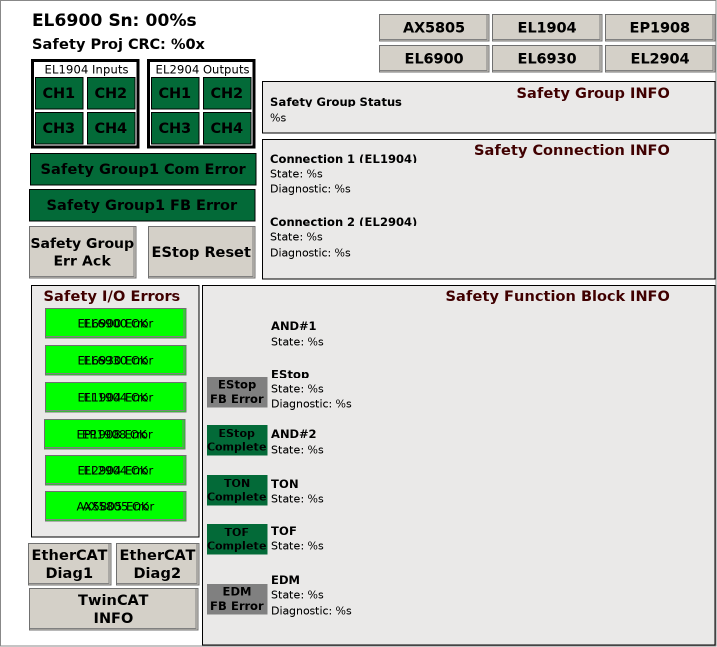
VISUALIZATION TwinSAFE  // 717x647
    RoundedRectangle (31,285 168x252)
    Rectangle (31,59 108x89)
    Rectangle (29,9 219x22), "EL6900 Sn: 00%s", text variable: g_udiHMI_SerialNumber
    Rectangle (29,33 232x22), "Safety Proj CRC: %0x", text variable: g_uiHMI_ProjectCRC
    Rectangle (35,77 48x32), "CH1", colour toggle: g_xHMI_EL1904Ch1
    Rectangle (87,77 48x32), "CH2", colour toggle: g_xHMI_EL1904Ch2
    Rectangle (35,112 48x32), "CH3", colour toggle: g_xHMI_EL1904Ch3
    Rectangle (87,112 48x32), "CH4", colour toggle: g_xHMI_EL1904Ch4
    Label (37,58 99x23), "EL1904 Inputs"
    Rectangle (147,59 108x89)
    Rectangle (151,77 48x32), "CH1", colour toggle: g_xHMI_EL2904Ch1
    Rectangle (203,77 48x32), "CH2", colour toggle: g_xHMI_EL2904Ch2
    Rectangle (151,112 48x32), "CH3", colour toggle: g_xHMI_EL2904Ch3
    Rectangle (203,112 48x32), "CH4", colour toggle: g_xHMI_EL2904Ch4
    Label (153,58 99x23), "EL2904 Outputs"
    Button (29,226 107x52), "Safety Group Err Ack"
        OnMouseDown: execute { g_xHMI_ErrAckPB := TRUE ; }
        OnMouseUp: execute { g_xHMI_ErrAckPB := FALSE ; }
    Button (148,226 107x52), "EStop Reset"
        OnMouseDown: execute { g_xHMI_EStopResetPB := TRUE ; }
        OnMouseUp: execute { g_xHMI_EStopResetPB := FALSE ; }
    Rectangle (30,153 226x32), "Safety Group1 Com Error", colour toggle: g_xHMI_SafetyGroup1_COMerrorLT
    Rectangle (29,189 226x32), "Safety Group1 FB Error", colour toggle: g_xHMI_SafetyGroup1_FBerrorLT
    Label (50,283 133x26), "Safety I/O Errors"
    Button (28,543 83x42), "EtherCAT Diag1"
        OnMouseClick: change screen: EtherCAT_Diag1
    Button (116,543 83x42), "EtherCAT Diag2"
        OnMouseClick: change screen: EtherCAT_Diag2
    Button (29,588 169x42), "TwinCAT INFO"
        OnMouseClick: change screen: TwinCAT_INFO
    RoundedRectangle (262,81 453x52)
    Label (449,80 224x26), "Safety Group INFO"
    Label (267,89 135x26), "Safety Group Status"
    RoundedRectangle (262,139 453x140)
    Label (449,137 224x26), "Safety Connection INFO"
    Label (267,146 203x26), "Connection 1 (EL1904)"
    Label (267,209 203x26), "Connection 2 (EL2904)"
    RoundedRectangle (202,285 513x360)
    Label (449,283 224x26), "Safety Function Block INFO"
    Label (268,313 50x26), "AND#1"
    Label (268,362 51x25), "EStop"
    Button (379,14 110x27), "AX5805"
        OnMouseClick: change screen: AX5805_Specific_Diagnostics
    Button (379,45 110x27), "EL6900"
        OnMouseClick: change screen: EL6900_Specific_Diagnostics
    Button (492,14 110x27), "EL1904"
        OnMouseClick: change screen: EL1904_Specific_Diagnostics
    Button (492,45 110x27), "EL6930"
        OnMouseClick: change screen: EL6930_Specific_Diagnostics
    Button (605,14 110x27), "EP1908"
        OnMouseClick: change screen: EP1908_Specific_Diagnostics
    Button (605,45 110x27), "EL2904"
        OnMouseClick: change screen: EL2904_Specific_Diagnostics
    Rectangle (267,107 321x22), "%s", text variable: g_sHMI_StatusGroup1
    Rectangle (267,163 321x22), "State: %s", text variable: g_sHMI_StateConn1
    Rectangle (267,178 386x22), "Diagnostic: %s", text variable: g_sHMI_DiagConn1
    Rectangle (267,226 321x22), "State: %s", text variable: g_sHMI_StateConn2
    Rectangle (267,242 389x22), "Diagnostic: %s", text variable: g_sHMI_DiagConn2
    Rectangle (268,331 439x22), "State: %s", text variable: g_sHMI_StatusAND1
    Rectangle (268,378 439x22), "State: %s", text variable: g_sHMI_StatusEStop1
    Rectangle (268,393 439x22), "Diagnostic: %s", text variable: g_sHMI_DiagEStop1
    Rectangle (268,439 439x22), "State: %s", text variable: g_sHMI_StatusAND2
    Label (268,421 54x26), "AND#2"
    Rectangle (268,488 439x22), "State: %s", text variable: g_sHMI_StatusTON
    Label (268,471 36x26), "TON"
    Rectangle (268,535 439x22), "State: %s", text variable: g_sHMI_StatusTOF
    Label (268,518 33x26), "TOF"
    Label (268,571 34x18), "EDM"
    Rectangle (268,584 439x22), "State: %s", text variable: g_sHMI_StatusEDM
    Rectangle (268,600 439x22), "Diagnostic: %s", text variable: g_sHMI_DiagEDM
    Rectangle (207,377 60x30), "EStop FB Error", colour toggle: g_xHMI_EStop_errorLT
    Rectangle (207,425 60x30), "EStop Complete", colour toggle: g_xHMI_EStop_CompleteLT
    Rectangle (207,475 60x30), "TON Complete", colour toggle: g_xHMI_EStop_ON_Delay_CompleteLT
    Rectangle (207,524 60x30), "TOF Complete", colour toggle: g_xHMI_EStop_OFF_Delay_CompleteLT
    Rectangle (207,584 60x30), "EDM FB Error", colour toggle: g_xHMI_EDMerrorLT
    Group (45,308 141x30)
        Button (0,0 141x30), colour toggle: g_xHMI_EL6900_General_Error
            OnMouseClick: change screen: AX5805_Specific_Diagnostics
            OnMouseUp: execute { g_xHMI_ErrAckPB := FALSE ; }
        Label (10,3 121x25), "EL6900 Error", invisible if: NOT g_xHMI_EL6900_General_Error
        Label (10,3 121x25), "EL6900 OK", invisible if: g_xHMI_EL6900_General_Error
    Group (45,345 141x30)
        Button (0,0 141x30), colour toggle: g_xHMI_EL6930_General_Error
            OnMouseClick: change screen: AX5805_Specific_Diagnostics
            OnMouseUp: execute { g_xHMI_ErrAckPB := FALSE ; }
        Label (10,3 121x25), "EL6930 Error", invisible if: NOT g_xHMI_EL6930_General_Error
        Label (10,3 121x25), "EL6930 OK", invisible if: g_xHMI_EL6930_General_Error
    Group (45,382 141x30)
        Button (0,0 141x30), colour toggle: g_xHMI_EL1904_General_Error
            OnMouseClick: change screen: AX5805_Specific_Diagnostics
            OnMouseUp: execute { g_xHMI_ErrAckPB := FALSE ; }
        Label (10,3 121x25), "EL1904 Error", invisible if: NOT g_xHMI_EL1904_General_Error
        Label (10,3 121x25), "EL1904 OK", invisible if: g_xHMI_EL1904_General_Error
    Group (44,419 141x30)
        Button (0,0 141x30), colour toggle: g_xHMI_EP1908_General_Error
            OnMouseClick: change screen: AX5805_Specific_Diagnostics
            OnMouseUp: execute { g_xHMI_ErrAckPB := FALSE ; }
        Label (10,3 121x25), "EP1908 Error", invisible if: NOT g_xHMI_EP1908_General_Error
        Label (10,3 121x25), "EP1908 OK", invisible if: g_xHMI_EP1908_General_Error
    Group (45,455 141x30)
        Button (0,0 141x30), colour toggle: g_xHMI_EL2904_General_Error
            OnMouseClick: change screen: AX5805_Specific_Diagnostics
            OnMouseUp: execute { g_xHMI_ErrAckPB := FALSE ; }
        Label (10,3 121x25), "EL2904 Error", invisible if: NOT g_xHMI_EL2904_General_Error
        Label (10,3 121x25), "EL2904 OK", invisible if: g_xHMI_EL2904_General_Error
    Group (45,491 141x30)
        Button (0,0 141x30), colour toggle: g_xHMI_AX5805_General_Error
            OnMouseClick: change screen: AX5805_Specific_Diagnostics
            OnMouseUp: execute { g_xHMI_ErrAckPB := FALSE ; }
        Label (10,3 121x25), "AX5805 Error", invisible if: NOT g_xHMI_AX5805_General_Error
        Label (10,3 121x25), "AX5805 OK", invisible if: g_xHMI_AX5805_General_Error
END_VISUALIZATION

// ---- VISUs/TwinSAFE.TcVIS
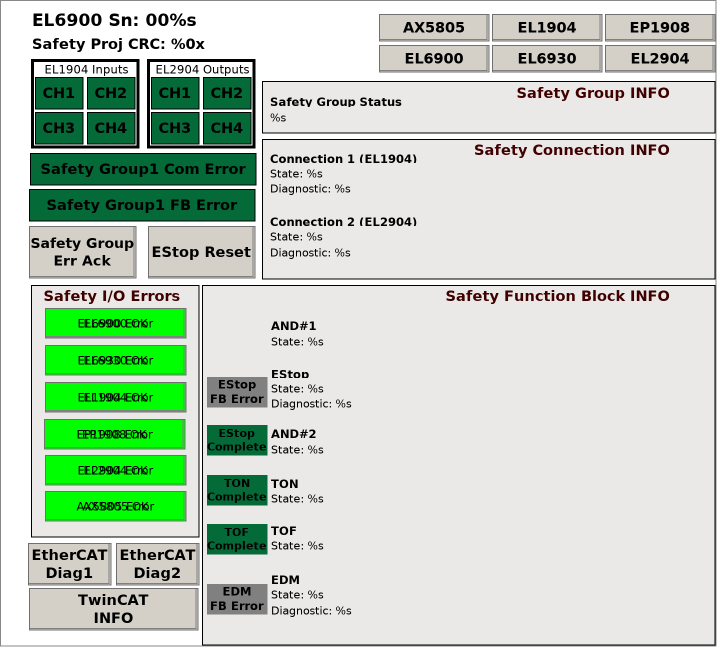
VISUALIZATION TwinSAFE  // 717x647
    RoundedRectangle (31,285 168x252)
    Rectangle (31,59 108x89)
    Rectangle (29,9 219x22), "EL6900 Sn: 00%s", text variable: g_udiHMI_SerialNumber
    Rectangle (29,33 232x22), "Safety Proj CRC: %0x", text variable: g_uiHMI_ProjectCRC
    Rectangle (35,77 48x32), "CH1", colour toggle: g_xHMI_EL1904Ch1
    Rectangle (87,77 48x32), "CH2", colour toggle: g_xHMI_EL1904Ch2
    Rectangle (35,112 48x32), "CH3", colour toggle: g_xHMI_EL1904Ch3
    Rectangle (87,112 48x32), "CH4", colour toggle: g_xHMI_EL1904Ch4
    Label (37,58 99x23), "EL1904 Inputs"
    Rectangle (147,59 108x89)
    Rectangle (151,77 48x32), "CH1", colour toggle: g_xHMI_EL2904Ch1
    Rectangle (203,77 48x32), "CH2", colour toggle: g_xHMI_EL2904Ch2
    Rectangle (151,112 48x32), "CH3", colour toggle: g_xHMI_EL2904Ch3
    Rectangle (203,112 48x32), "CH4", colour toggle: g_xHMI_EL2904Ch4
    Label (153,58 99x23), "EL2904 Outputs"
    Button (29,226 107x52), "Safety Group Err Ack"
        OnMouseDown: execute { g_xHMI_ErrAckPB := TRUE ; }
        OnMouseUp: execute { g_xHMI_ErrAckPB := FALSE ; }
    Button (148,226 107x52), "EStop Reset"
        OnMouseDown: execute { g_xHMI_EStopResetPB := TRUE ; }
        OnMouseUp: execute { g_xHMI_EStopResetPB := FALSE ; }
    Rectangle (30,153 226x32), "Safety Group1 Com Error", colour toggle: g_xHMI_SafetyGroup1_COMerrorLT
    Rectangle (29,189 226x32), "Safety Group1 FB Error", colour toggle: g_xHMI_SafetyGroup1_FBerrorLT
    Label (50,283 133x26), "Safety I/O Errors"
    Button (28,543 83x42), "EtherCAT Diag1"
        OnMouseClick: change screen: EtherCAT_Diag1
    Button (116,543 83x42), "EtherCAT Diag2"
        OnMouseClick: change screen: EtherCAT_Diag2
    Button (29,588 169x42), "TwinCAT INFO"
        OnMouseClick: change screen: TwinCAT_INFO
    RoundedRectangle (262,81 453x52)
    Label (449,80 224x26), "Safety Group INFO"
    Label (267,89 135x26), "Safety Group Status"
    RoundedRectangle (262,139 453x140)
    Label (449,137 224x26), "Safety Connection INFO"
    Label (267,146 203x26), "Connection 1 (EL1904)"
    Label (267,209 203x26), "Connection 2 (EL2904)"
    RoundedRectangle (202,285 513x360)
    Label (449,283 224x26), "Safety Function Block INFO"
    Label (268,313 50x26), "AND#1"
    Label (268,362 51x25), "EStop"
    Button (379,14 110x27), "AX5805"
        OnMouseClick: change screen: AX5805_Specific_Diagnostics
    Button (379,45 110x27), "EL6900"
        OnMouseClick: change screen: EL6900_Specific_Diagnostics
    Button (492,14 110x27), "EL1904"
        OnMouseClick: change screen: EL1904_Specific_Diagnostics
    Button (492,45 110x27), "EL6930"
        OnMouseClick: change screen: EL6930_Specific_Diagnostics
    Button (605,14 110x27), "EP1908"
        OnMouseClick: change screen: EP1908_Specific_Diagnostics
    Button (605,45 110x27), "EL2904"
        OnMouseClick: change screen: EL2904_Specific_Diagnostics
    Rectangle (267,107 321x22), "%s", text variable: g_sHMI_StatusGroup1
    Rectangle (267,163 321x22), "State: %s", text variable: g_sHMI_StateConn1
    Rectangle (267,178 386x22), "Diagnostic: %s", text variable: g_sHMI_DiagConn1
    Rectangle (267,226 321x22), "State: %s", text variable: g_sHMI_StateConn2
    Rectangle (267,242 389x22), "Diagnostic: %s", text variable: g_sHMI_DiagConn2
    Rectangle (268,331 439x22), "State: %s", text variable: g_sHMI_StatusAND1
    Rectangle (268,378 439x22), "State: %s", text variable: g_sHMI_StatusEStop1
    Rectangle (268,393 439x22), "Diagnostic: %s", text variable: g_sHMI_DiagEStop1
    Rectangle (268,439 439x22), "State: %s", text variable: g_sHMI_StatusAND2
    Label (268,421 54x26), "AND#2"
    Rectangle (268,488 439x22), "State: %s", text variable: g_sHMI_StatusTON
    Label (268,471 36x26), "TON"
    Rectangle (268,535 439x22), "State: %s", text variable: g_sHMI_StatusTOF
    Label (268,518 33x26), "TOF"
    Label (268,571 34x18), "EDM"
    Rectangle (268,584 439x22), "State: %s", text variable: g_sHMI_StatusEDM
    Rectangle (268,600 439x22), "Diagnostic: %s", text variable: g_sHMI_DiagEDM
    Rectangle (207,377 60x30), "EStop FB Error", colour toggle: g_xHMI_EStop_errorLT
    Rectangle (207,425 60x30), "EStop Complete", colour toggle: g_xHMI_EStop_CompleteLT
    Rectangle (207,475 60x30), "TON Complete", colour toggle: g_xHMI_EStop_ON_Delay_CompleteLT
    Rectangle (207,524 60x30), "TOF Complete", colour toggle: g_xHMI_EStop_OFF_Delay_CompleteLT
    Rectangle (207,584 60x30), "EDM FB Error", colour toggle: g_xHMI_EDMerrorLT
    Group (45,308 141x30)
        Button (0,0 141x30), colour toggle: g_xHMI_EL6900_General_Error
            OnMouseClick: change screen: AX5805_Specific_Diagnostics
            OnMouseUp: execute { g_xHMI_ErrAckPB := FALSE ; }
        Label (10,3 121x25), "EL6900 Error", invisible if: NOT g_xHMI_EL6900_General_Error
        Label (10,3 121x25), "EL6900 OK", invisible if: g_xHMI_EL6900_General_Error
    Group (45,345 141x30)
        Button (0,0 141x30), colour toggle: g_xHMI_EL6930_General_Error
            OnMouseClick: change screen: AX5805_Specific_Diagnostics
            OnMouseUp: execute { g_xHMI_ErrAckPB := FALSE ; }
        Label (10,3 121x25), "EL6930 Error", invisible if: NOT g_xHMI_EL6930_General_Error
        Label (10,3 121x25), "EL6930 OK", invisible if: g_xHMI_EL6930_General_Error
    Group (45,382 141x30)
        Button (0,0 141x30), colour toggle: g_xHMI_EL1904_General_Error
            OnMouseClick: change screen: AX5805_Specific_Diagnostics
            OnMouseUp: execute { g_xHMI_ErrAckPB := FALSE ; }
        Label (10,3 121x25), "EL1904 Error", invisible if: NOT g_xHMI_EL1904_General_Error
        Label (10,3 121x25), "EL1904 OK", invisible if: g_xHMI_EL1904_General_Error
    Group (44,419 141x30)
        Button (0,0 141x30), colour toggle: g_xHMI_EP1908_General_Error
            OnMouseClick: change screen: AX5805_Specific_Diagnostics
            OnMouseUp: execute { g_xHMI_ErrAckPB := FALSE ; }
        Label (10,3 121x25), "EP1908 Error", invisible if: NOT g_xHMI_EP1908_General_Error
        Label (10,3 121x25), "EP1908 OK", invisible if: g_xHMI_EP1908_General_Error
    Group (45,455 141x30)
        Button (0,0 141x30), colour toggle: g_xHMI_EL2904_General_Error
            OnMouseClick: change screen: AX5805_Specific_Diagnostics
            OnMouseUp: execute { g_xHMI_ErrAckPB := FALSE ; }
        Label (10,3 121x25), "EL2904 Error", invisible if: NOT g_xHMI_EL2904_General_Error
        Label (10,3 121x25), "EL2904 OK", invisible if: g_xHMI_EL2904_General_Error
    Group (45,491 141x30)
        Button (0,0 141x30), colour toggle: g_xHMI_AX5805_General_Error
            OnMouseClick: change screen: AX5805_Specific_Diagnostics
            OnMouseUp: execute { g_xHMI_ErrAckPB := FALSE ; }
        Label (10,3 121x25), "AX5805 Error", invisible if: NOT g_xHMI_AX5805_General_Error
        Label (10,3 121x25), "AX5805 OK", invisible if: g_xHMI_AX5805_General_Error
END_VISUALIZATION
